// TwinCAT 3 PLC project Library
// Title: lcls-twincat-common-components
// Company: SLAC
// ProjectVersion: 4.0.0
// ProgramVersion: 3.1.4026.17
// libraries:
//   LCLS General, * (SLAC)
//   LCLS_Tc_Motion, * (SLAC - LCLS)
//   LCLS_Tc_DevAbs, * (SLAC - LCLS)
//   lcls-twincat-physics, * (SLAC)
//   PMPS, * (SLAC - LCLS)
//   Tc2_MC2, * (Beckhoff Automation GmbH)
//   Tc2_SerialCom, * (Beckhoff Automation GmbH)
//   Tc2_Standard, * (Beckhoff Automation GmbH)
//   Tc2_Utilities, * (Beckhoff Automation GmbH)
//   Tc3_JsonXml, * (Beckhoff Automation GmbH)
//   Tc3_Module, * (Beckhoff Automation GmbH)
//   TcUnit, * (www.tcunit.org)
// project tree:
//   Devices/ATM/ E_ATM_States.TcDUT, FB_ATM.TcPOU
//   Devices/LIC/ E_LIC_States.TcDUT, FB_LIC.TcPOU
//   Devices/PPM/ E_PPM_States.TcDUT, FB_PPM.TcPOU, FB_PPM_Gige.TcPOU, FB_PPM_PowerMeter.TcPOU
//   Devices/REF/ E_REF_States.TcDUT, FB_REF.TcPOU, FB_REF_Laser.TcPOU
//   Devices/SATT/ E_SXR_SATT_Position.TcDUT, FB_AttenuatorElementDensity.TcPOU, FB_SATT_FilterConfig.TcPOU, FB_SXR_SATT_Stage.TcPOU, ST_SATT_Filter.TcDUT
//   Devices/SLITS/ E_SlitsBlade.TcDUT, FB_SLITS.TcPOU, FB_SLITS_POWER.TcPOU
//   Devices/WFS/ E_WFS_States.TcDUT, FB_WFS.TcPOU
//   Devices/GBS/ E_GBS_States.TcDUT, FB_GBS.TcPOU
//   Devices/IPM/ E_IPM_States.TcDUT, FB_IPM.TcPOU
//   Devices/XPIM/ E_XPIM_Filters.TcDUT, E_XPIM_States.TcDUT, FB_XPIM.TcPOU, FB_XPIM_FilterWheel.TcPOU, FB_XPIM_LED.TcPOU, FB_XPIM_Opal.TcPOU
//   / PlcTask.TcTTO
//   POUs/ FB_CC_TempSensor.TcPOU, FB_CC_InternalStateConfig.TcPOU, FB_CC_StateDefaultsConfig.TcPOU, FB_CC_StatePMPSConfig.TcPOU, FB_FDQ_FlowMeter.TcPOU, FB_XTES_Flowswitch.TcPOU
//   Tests/ FB_ATMTest.TcPOU, FB_CC_TempSensorTest.TcPOU, FB_GBSTest.TcPOU, FB_IPMTest.TcPOU, FB_SATTTest.TcPOU, FB_LICTest.TcPOU, FB_PPMTest.TcPOU, FB_REFTest.TcPOU, FB_SLITS_POWERTest.TcPOU, FB_WFSTest.TcPOU, FB_XPIMTest.TcPOU, PRG_TEST.TcPOU
//   Tests/Helpers/ FB_PMPSJsonTestHelper.TcPOU, FB_CC_PMPSTestSetup.TcPOU
//   Version/ Global_Version.TcGVL
// real-time tasks:
//   TASK PlcTask: cycle T#10ms, priority 20, ADS port 350
// motion (NC):
//   TASK NC-Task 1 SAF: cycle T#2ms, priority 4, ADS port 501
//   TASK NC-Task 1 SVB: cycle T#10ms, priority 8, ADS port 511
//   AXIS IPM_Y (id 13)
//   AXIS GBS_Y (id 12)
//   AXIS ATM_Y (id 1)
//     OtherSettings: AllowMotionCmdToSlave=true
//     encoder EncType=1
//     drive DrvType=5
//       Analog: TorqueSetpointScale=10, ScaleFactorActTorque=0.1
//       TimeComp: TaskDelayCycles=1
//     controller CtrType=1
//       CtrPara: PriorControlFactor=1
//         Observer: BandWidth=20
//   AXIS LIC_Y (id 2)
//     OtherSettings: AllowMotionCmdToSlave=true
//     encoder EncType=1
//     drive DrvType=5
//       Analog: TorqueSetpointScale=10, ScaleFactorActTorque=0.1
//       TimeComp: TaskDelayCycles=1
//     controller CtrType=1
//       CtrPara: PriorControlFactor=1
//         Observer: BandWidth=20
//   AXIS PPM_Y (id 3)
//     OtherSettings: AllowMotionCmdToSlave=true
//     encoder EncType=1
//     drive DrvType=5
//       Analog: TorqueSetpointScale=10, ScaleFactorActTorque=0.1
//       TimeComp: TaskDelayCycles=1
//     controller CtrType=1
//       CtrPara: PriorControlFactor=1
//         Observer: BandWidth=20
//   AXIS REF_Y (id 4)
//     OtherSettings: AllowMotionCmdToSlave=true
//     encoder EncType=1
//     drive DrvType=5
//       Analog: TorqueSetpointScale=10, ScaleFactorActTorque=0.1
//       TimeComp: TaskDelayCycles=1
//     controller CtrType=1
//       CtrPara: PriorControlFactor=1
//         Observer: BandWidth=20
//   AXIS SATT_Y (id 7)
//     OtherSettings: AllowMotionCmdToSlave=true
//     encoder EncType=1
//     drive DrvType=5
//       Analog: TorqueSetpointScale=10, ScaleFactorActTorque=0.1
//     controller CtrType=1
//       CtrPara: PriorControlFactor=1
//         Observer: BandWidth=20
//   AXIS WFS_Y (id 5)
//     OtherSettings: AllowMotionCmdToSlave=true
//     encoder EncType=1
//     drive DrvType=5
//       Analog: TorqueSetpointScale=10, ScaleFactorActTorque=0.1
//       TimeComp: TaskDelayCycles=1
//     controller CtrType=1
//       CtrPara: PriorControlFactor=1
//         Observer: BandWidth=20
//   AXIS XPIM_Y (id 6)
//     OtherSettings: AllowMotionCmdToSlave=true
//     encoder EncType=1
//     drive DrvType=5
//       Analog: TorqueSetpointScale=10, ScaleFactorActTorque=0.1
//       TimeComp: TaskDelayCycles=1
//     controller CtrType=1
//       CtrPara: PriorControlFactor=1
//         Observer: BandWidth=20
//   AXIS SLIT_Bottom (id 9)
//   AXIS SLIT_North (id 10)
//   AXIS SLIT_South (id 11)
//   AXIS SLIT_Top (id 8)
//     OtherSettings: AllowMotionCmdToSlave=true
//     encoder EncType=1
//     drive DrvType=5
//       Analog: TorqueSetpointScale=10, ScaleFactorActTorque=0.1
//       TimeComp: TaskDelayCycles=1
//     controller CtrType=1
//       CtrPara: PriorControlFactor=1
//         Observer: BandWidth=20
// variable links:
//   Library Instance <-> NC-Task 1 SAF/Axes/ATM_Y
//     PlcTask Inputs/PRG_TEST.fbATMTest.axRef[2].NcToPlc <-> Outputs/ToPlc
//     PlcTask Outputs/PRG_TEST.fbATMTest.axRef[2].PlcToNc <-> Inputs/FromPlc
//   Library Instance <-> NC-Task 1 SAF/Axes/GBS_Y
//     PlcTask Inputs/PRG_TEST.fbGBSTest.axRef.NcToPlc <-> Outputs/ToPlc
//     PlcTask Outputs/PRG_TEST.fbGBSTest.axRef.PlcToNc <-> Inputs/FromPlc
//   Library Instance <-> NC-Task 1 SAF/Axes/IPM_Y
//     PlcTask Inputs/PRG_TEST.fbIPMTest.axRef[2].NcToPlc <-> Outputs/ToPlc
//     PlcTask Outputs/PRG_TEST.fbIPMTest.axRef[2].PlcToNc <-> Inputs/FromPlc
//   Library Instance <-> NC-Task 1 SAF/Axes/LIC_Y
//     PlcTask Inputs/PRG_TEST.fbLICTest.axRef.NcToPlc <-> Outputs/ToPlc
//     PlcTask Outputs/PRG_TEST.fbLICTest.axRef.PlcToNc <-> Inputs/FromPlc
//   Library Instance <-> NC-Task 1 SAF/Axes/PPM_Y
//     PlcTask Inputs/PRG_TEST.fbPPMTest.axRef.NcToPlc <-> Outputs/ToPlc
//     PlcTask Outputs/PRG_TEST.fbPPMTest.axRef.PlcToNc <-> Inputs/FromPlc
//   Library Instance <-> NC-Task 1 SAF/Axes/REF_Y
//     PlcTask Inputs/PRG_TEST.fbREFTest.axRef[2].NcToPlc <-> Outputs/ToPlc
//     PlcTask Outputs/PRG_TEST.fbREFTest.axRef[2].PlcToNc <-> Inputs/FromPlc
//   Library Instance <-> NC-Task 1 SAF/Axes/SATT_Y
//     PlcTask Inputs/PRG_TEST.fbSATTTest.axRef.NcToPlc <-> Outputs/ToPlc
//     PlcTask Outputs/PRG_TEST.fbSATTTest.axRef.PlcToNc <-> Inputs/FromPlc
//   Library Instance <-> NC-Task 1 SAF/Axes/SLIT_Bottom
//     PlcTask Inputs/PRG_TEST.fbSlitsPowerTest.axRef[2].NcToPlc <-> Outputs/ToPlc
//     PlcTask Outputs/PRG_TEST.fbSlitsPowerTest.axRef[2].PlcToNc <-> Inputs/FromPlc
//   Library Instance <-> NC-Task 1 SAF/Axes/SLIT_North
//     PlcTask Inputs/PRG_TEST.fbSlitsPowerTest.axRef[3].NcToPlc <-> Outputs/ToPlc
//     PlcTask Outputs/PRG_TEST.fbSlitsPowerTest.axRef[3].PlcToNc <-> Inputs/FromPlc
//   Library Instance <-> NC-Task 1 SAF/Axes/SLIT_South
//     PlcTask Inputs/PRG_TEST.fbSlitsPowerTest.axRef[4].NcToPlc <-> Outputs/ToPlc
//     PlcTask Outputs/PRG_TEST.fbSlitsPowerTest.axRef[4].PlcToNc <-> Inputs/FromPlc
//   Library Instance <-> NC-Task 1 SAF/Axes/SLIT_Top
//     PlcTask Inputs/PRG_TEST.fbSlitsPowerTest.axRef[1].NcToPlc <-> Outputs/ToPlc
//     PlcTask Outputs/PRG_TEST.fbSlitsPowerTest.axRef[1].PlcToNc <-> Inputs/FromPlc
//   Library Instance <-> NC-Task 1 SAF/Axes/WFS_Y
//     PlcTask Inputs/PRG_TEST.fbWFSTest.axRef[2].NcToPlc <-> Outputs/ToPlc
//     PlcTask Outputs/PRG_TEST.fbWFSTest.axRef[2].PlcToNc <-> Inputs/FromPlc
//   Library Instance <-> NC-Task 1 SAF/Axes/XPIM_Y
//     PlcTask Inputs/PRG_TEST.fbXPIMTest.axRef[3].NcToPlc <-> Outputs/ToPlc
//     PlcTask Outputs/PRG_TEST.fbXPIMTest.axRef[3].PlcToNc <-> Inputs/FromPlc

CONFIGURATION Library
    RESOURCE PLC ON TwinCAT3
        TASK PlcTask(INTERVAL := T#10ms, PRIORITY := 20);
        PROGRAM PRG_TEST WITH PlcTask : PRG_TEST;
    END_RESOURCE
END_CONFIGURATION

// ---- Devices/ATM/E_ATM_States.TcDUT
{attribute 'qualified_only'}
TYPE E_ATM_States :
(
    Unknown := 0,
    OUT := 1,
    TARGET1 := 2,
    TARGET2 := 3,
    TARGET3 := 4,
    TARGET4 := 5,
    TARGET5 := 6,
    TARGET6 := 7,
    TARGET7 := 8
) UINT;
END_TYPE

// ---- Devices/LIC/E_LIC_States.TcDUT
{attribute 'qualified_only'}
TYPE E_LIC_States :
(
    Unknown := 0,
    OUT := 1,
    MIRROR1 := 2,
    MIRROR2 := 3,
    TARGET := 4
) UINT;
END_TYPE

// ---- Devices/PPM/E_PPM_States.TcDUT
{attribute 'qualified_only'}
TYPE E_PPM_States :
(
    Unknown := 0,
    OUT := 1,
    POWERMETER := 2,
    YAG1 := 3,
    YAG2 := 4
) UINT;
END_TYPE

// ---- Devices/REF/E_REF_States.TcDUT
(* REF state-select enum. UINT-typed so REFERENCE TO E_REF_States
   is bridge-compatible with the ND mover's REFERENCE TO UINT. *)
{attribute 'qualified_only'}
{attribute 'strict'}
TYPE E_REF_States :
(
    UNKNOWN := 0,
    OUT     := 1,
    IN      := 2
) UINT;
END_TYPE

// ---- Devices/SATT/E_SXR_SATT_Position.TcDUT
{attribute 'qualified_only'}
TYPE E_SXR_SATT_Position :
(
    UNKNOWN := 0, // UNKNOWN must be in slot 0 or the FB breaks
    OUT := 1, // OUT at slot 1 is a convention
    FILTER1 := 2,
    FILTER2 := 3,
    FILTER3 := 4,
    FILTER4 := 5,
    FILTER5 := 6,
    FILTER6 := 7,
    FILTER7 := 8,
    FILTER8 := 9
) UINT;
END_TYPE

// ---- Devices/SATT/ST_SATT_Filter.TcDUT
TYPE ST_SATT_Filter :
STRUCT
    {attribute 'pytmc' := '
        pv: MATERIAL
        io: input
        field: DESC Filter material name
    '}
    sFilterMaterial : STRING;

    {attribute 'pytmc' := '
        pv: THICKNESS
        io: input
        field: DESC Filter material thickness
        field: EGU um
    '}
    fFilterThickness_um : LREAL;
END_STRUCT
END_TYPE

// ---- Devices/SLITS/E_SlitsBlade.TcDUT
(* Blade index into the four-element slit motion-stage array
   (Top / Bottom / North / South). Values 1..4 match the array bounds. *)
{attribute 'qualified_only'}
{attribute 'strict'}
TYPE E_SlitsBlade :
(
    TOP    := 1,
    BOTTOM := 2,
    NORTH  := 3,
    SOUTH  := 4
) UDINT;
END_TYPE

// ---- Devices/WFS/E_WFS_States.TcDUT
{attribute 'qualified_only'}
TYPE E_WFS_States :
(
    Unknown := 0,
    OUT := 1,
    TARGET1 := 2,
    TARGET2 := 3,
    TARGET3 := 4,
    TARGET4 := 5,
    TARGET5 := 6
) UINT;
END_TYPE

// ---- Devices/GBS/E_GBS_States.TcDUT
{attribute 'qualified_only'}
TYPE E_GBS_States :
(
    Unknown := 0,
    OUT := 1,
    TARGET1a := 2,
    TARGET1b := 3,
    TARGET2a := 4,
    TARGET2b := 5,
    TARGET3a := 6,
    TARGET3b := 7,
    TARGET4 := 8,
    TARGET5 := 9,
    TARGET6 := 10
) UINT;
END_TYPE

// ---- Devices/IPM/E_IPM_States.TcDUT
{attribute 'qualified_only'}
TYPE E_IPM_States :
(
    Unknown := 0,
    OUT := 1,
    TARGET1 := 2,
    TARGET2 := 3,
    TARGET3 := 4,
    TARGET4 := 5
) UINT;
END_TYPE

// ---- Devices/XPIM/E_XPIM_Filters.TcDUT
{attribute 'qualified_only'}
TYPE E_XPIM_Filters :
(
    Unknown := 0,
    T50 := 1,
    T25 := 2,
    T10 := 3,
    T5 := 4,
    T1 := 5,
    T100 := 6
) UINT;
END_TYPE

// ---- Devices/XPIM/E_XPIM_States.TcDUT
{attribute 'qualified_only'}
TYPE E_XPIM_States :
(
    Unknown := 0,
    OUT := 1,
    YAG := 2,
    DIAMOND := 3,
    RETICLE := 4
) UINT;
END_TYPE

// ---- Version/Global_Version.TcGVL
{attribute 'TcGenerated'}
{attribute 'no-analysis'}
{attribute 'linkalways'}
// This function has been automatically generated from the project information.
VAR_GLOBAL CONSTANT
    {attribute 'const_non_replaced'}
    stLibVersion_lcls_twincat_common_components : ST_LibVersion := (iMajor := 4, iMinor := 0, iBuild := 0, iRevision := 0, nFlags := 1, sVersion := '4.0.0');
END_VAR

// ---- Tests/PRG_TEST.TcPOU
{attribute 'analysis' := '-33'}
PROGRAM PRG_TEST
VAR
    (* Seeds PMPS_GVL.BP_jsonDoc with the fake test PMPS DB in before any test FB body runs. *)
    fbPmpsTestSetup: FB_CC_PMPSTestSetup;
    fbATMTest: FB_ATMTest;
    fbGBSTest: FB_GBSTest;
    fbIPMTest: FB_IPMTest;
    fbLICTest: FB_LICTest;
    fbPPMTest: FB_PPMTest;
    fbREFTest: FB_REFTest;
    fbSATTTest: FB_SATTTest;
    fbSlitsPowerTest: FB_SLITS_POWERTest;
    fbWFSTest: FB_WFSTest;
    fbXPIMTest: FB_XPIMTest;
    fbCCTempSensorTest: FB_CC_TempSensorTest;


END_VAR

// Run the tests
TcUnit.RUN();

END_PROGRAM

// ---- Tests/Helpers/FB_CC_PMPSTestSetup.TcPOU

(*
    One-shot PMPS fake-DB seeder for the CC test suite. Mirrors
    LCLS_Tc_Motion.FB_PMPSTestSetup: one FB_PMPSJsonTestHelperEx
    instance per device, first call uses bNewDoc := TRUE, the rest
    use bNewDoc := FALSE so the document at PMPS_GVL.BP_jsonDoc
    accumulates every test device:

        { "TST:ATM": { "TST:ATM-TRANSITION": {...}, ... },
          "TST:LIC": { ... }, ... }

    Only sPmpsState is populated per row. The helper fills the rest
    of the JSON shape with default-zero values, which is enough for
    the wiring smoke tests to look up state keys and request a move.
    Tests that need richer beam params (rate, beam class, eV range,
    reactive temperature) set them on the relevant astParams_XXX
    entries before this FB ticks, or extend it.

    The seeding runs once in CallAfterInit, before any test suite
    body executes. The cyclic body is empty: no scheduling order
    dependency between this FB and the test FBs.

    Single point of truth: PMPS_GVL.BP_jsonDoc is global and test
    FBs run concurrently. Seeding stays here so per-device writes
    cannot race on the same cycle.
*)
{attribute 'call_after_init'}
{attribute 'analysis' := '-33'}
FUNCTION_BLOCK FB_CC_PMPSTestSetup
VAR
    (* All devices use the local FB_PMPSJsonTestHelper: it serializes the
       seeded nRequestAssertionID into the DB 'id' (so each state gets a
       unique assertion ID) and serializes nTempSP into reactive_temp
       (needed by SATT/SLITS RTD thresholds). *)
    fbJsonHelper_ATM   : FB_PMPSJsonTestHelper;
    fbJsonHelper_LIC   : FB_PMPSJsonTestHelper;
    fbJsonHelper_PPM   : FB_PMPSJsonTestHelper;
    fbJsonHelper_REF   : FB_PMPSJsonTestHelper;
    fbJsonHelper_GBS   : FB_PMPSJsonTestHelper;
    fbJsonHelper_IPM   : FB_PMPSJsonTestHelper;
    fbJsonHelper_WFS   : FB_PMPSJsonTestHelper;
    fbJsonHelper_XPIM  : FB_PMPSJsonTestHelper;
    fbJsonHelper_SATT  : FB_PMPSJsonTestHelper;
    fbJsonHelper_SLITS : FB_PMPSJsonTestHelper;

    (* astParams_XXX[0] is the transition key; the rest are named-state
       keys in enum order. *)
    astParams_ATM   : ARRAY[0..6] OF ST_DbStateParams;
    astParams_LIC   : ARRAY[0..4] OF ST_DbStateParams;
    astParams_PPM   : ARRAY[0..4] OF ST_DbStateParams;
    astParams_REF   : ARRAY[0..2] OF ST_DbStateParams;
    astParams_GBS   : ARRAY[0..10] OF ST_DbStateParams;
    astParams_IPM   : ARRAY[0..5] OF ST_DbStateParams;
    astParams_WFS   : ARRAY[0..6] OF ST_DbStateParams;
    astParams_XPIM  : ARRAY[0..5] OF ST_DbStateParams;
    astParams_SATT  : ARRAY[0..0] OF ST_DbStateParams;
    astParams_SLITS : ARRAY[0..0] OF ST_DbStateParams;
END_VAR


(* Seeding runs once at instantiation in CallAfterInit; body is a no-op. *)

{attribute 'call_after_init'}
METHOD CallAfterInit

(* ---- TST:ATM ---- *)
astParams_ATM[0].sPmpsState                  := 'TST:ATM-TRANSITION';
astParams_ATM[0].nRequestAssertionID         := 100;
astParams_ATM[0].stReactiveParams.nTempSP   := 30;
astParams_ATM[0].stBeamParams.nBeamClass     := 2#0000_1000;
astParams_ATM[0].stBeamParams.neVRange       := 2#1111_1111_1111_1111_1111_1111_1111_1111;
astParams_ATM[0].stBeamParams.nRate          := 1;
astParams_ATM[0].stBeamParams.nTran          := 0;
astParams_ATM[0].stBeamParams.nMachineMode   := 1;

astParams_ATM[1].sPmpsState                  := 'TST:ATM-OUT';
astParams_ATM[1].nRequestAssertionID         := 101;
astParams_ATM[1].stReactiveParams.nTempSP   := 30;
astParams_ATM[1].stBeamParams.nBeamClass     := 2#0000_0001;
astParams_ATM[1].stBeamParams.neVRange       := 2#1111_1111_1111_1111_1111_1111_1111_1111;
astParams_ATM[1].stBeamParams.nRate          := 10;
astParams_ATM[1].stBeamParams.nTran          := 12;
astParams_ATM[1].stBeamParams.nMachineMode   := 2;

astParams_ATM[2].sPmpsState                  := 'TST:ATM-TARGET1';
astParams_ATM[2].nRequestAssertionID         := 102;
astParams_ATM[2].stReactiveParams.nTempSP   := 30;
astParams_ATM[2].stBeamParams.nBeamClass     := 2#0000_0010;
astParams_ATM[2].stBeamParams.neVRange       := 2#1111_1111_1111_1111_1111_1111_1111_1111;
astParams_ATM[2].stBeamParams.nRate          := 50;
astParams_ATM[2].stBeamParams.nTran          := 8;
astParams_ATM[2].stBeamParams.nMachineMode   := 1;

astParams_ATM[3].sPmpsState                  := 'TST:ATM-TARGET2';
astParams_ATM[3].nRequestAssertionID         := 103;
astParams_ATM[3].stReactiveParams.nTempSP   := 30;
astParams_ATM[3].stBeamParams.nBeamClass     := 2#0000_0100;
astParams_ATM[3].stBeamParams.neVRange       := 2#1111_1111_1111_1111_1111_1111_1111_1111;
astParams_ATM[3].stBeamParams.nRate          := 50;
astParams_ATM[3].stBeamParams.nTran          := 8;
astParams_ATM[3].stBeamParams.nMachineMode   := 1;

astParams_ATM[4].sPmpsState                  := 'TST:ATM-TARGET3';
astParams_ATM[4].nRequestAssertionID         := 104;
astParams_ATM[4].stReactiveParams.nTempSP   := 30;
astParams_ATM[4].stBeamParams.nBeamClass     := 2#0001_0000;
astParams_ATM[4].stBeamParams.neVRange       := 2#1111_1111_1111_1111_1111_1111_1111_1111;
astParams_ATM[4].stBeamParams.nRate          := 50;
astParams_ATM[4].stBeamParams.nTran          := 8;
astParams_ATM[4].stBeamParams.nMachineMode   := 1;

astParams_ATM[5].sPmpsState                  := 'TST:ATM-TARGET4';
astParams_ATM[5].nRequestAssertionID         := 105;
astParams_ATM[5].stReactiveParams.nTempSP   := 30;
astParams_ATM[5].stBeamParams.nBeamClass     := 2#0010_0000;
astParams_ATM[5].stBeamParams.neVRange       := 2#1111_1111_1111_1111_1111_1111_1111_1111;
astParams_ATM[5].stBeamParams.nRate          := 50;
astParams_ATM[5].stBeamParams.nTran          := 8;
astParams_ATM[5].stBeamParams.nMachineMode   := 1;

astParams_ATM[6].sPmpsState                  := 'TST:ATM-TARGET5';
astParams_ATM[6].nRequestAssertionID         := 106;
astParams_ATM[6].stReactiveParams.nTempSP   := 30;
astParams_ATM[6].stBeamParams.nBeamClass     := 2#0100_0000;
astParams_ATM[6].stBeamParams.neVRange       := 2#1111_1111_1111_1111_1111_1111_1111_1111;
astParams_ATM[6].stBeamParams.nRate          := 50;
astParams_ATM[6].stBeamParams.nTran          := 8;
astParams_ATM[6].stBeamParams.nMachineMode   := 1;

(* ---- TST:LIC ---- *)
astParams_LIC[0].sPmpsState                  := 'TST:LIC-TRANSITION';
astParams_LIC[0].nRequestAssertionID         := 200;
astParams_LIC[0].stBeamParams.nBeamClass     := 2#0000_1000;
astParams_LIC[0].stBeamParams.neVRange       := 2#1111_1111_1111_1111_1111_1111_1111_1111;
astParams_LIC[0].stBeamParams.nRate          := 1;
astParams_LIC[0].stBeamParams.nTran          := 0;
astParams_LIC[0].stBeamParams.nMachineMode   := 1;

astParams_LIC[1].sPmpsState                  := 'TST:LIC-OUT';
astParams_LIC[1].nRequestAssertionID         := 201;
astParams_LIC[1].stBeamParams.nBeamClass     := 2#0000_0001;
astParams_LIC[1].stBeamParams.neVRange       := 2#1111_1111_1111_1111_1111_1111_1111_1111;
astParams_LIC[1].stBeamParams.nRate          := 10;
astParams_LIC[1].stBeamParams.nTran          := 12;
astParams_LIC[1].stBeamParams.nMachineMode   := 2;

astParams_LIC[2].sPmpsState                  := 'TST:LIC-MIRROR1';
astParams_LIC[2].nRequestAssertionID         := 202;
astParams_LIC[2].stBeamParams.nBeamClass     := 2#0000_0010;
astParams_LIC[2].stBeamParams.neVRange       := 2#1111_1111_1111_1111_1111_1111_1111_1111;
astParams_LIC[2].stBeamParams.nRate          := 50;
astParams_LIC[2].stBeamParams.nTran          := 8;
astParams_LIC[2].stBeamParams.nMachineMode   := 1;

astParams_LIC[3].sPmpsState                  := 'TST:LIC-MIRROR2';
astParams_LIC[3].nRequestAssertionID         := 203;
astParams_LIC[3].stBeamParams.nBeamClass     := 2#0000_0100;
astParams_LIC[3].stBeamParams.neVRange       := 2#1111_1111_1111_1111_1111_1111_1111_1111;
astParams_LIC[3].stBeamParams.nRate          := 50;
astParams_LIC[3].stBeamParams.nTran          := 8;
astParams_LIC[3].stBeamParams.nMachineMode   := 1;

astParams_LIC[4].sPmpsState                  := 'TST:LIC-TARGET';
astParams_LIC[4].nRequestAssertionID         := 204;
astParams_LIC[4].stBeamParams.nBeamClass     := 2#0001_0000;
astParams_LIC[4].stBeamParams.neVRange       := 2#1111_1111_1111_1111_1111_1111_1111_1111;
astParams_LIC[4].stBeamParams.nRate          := 50;
astParams_LIC[4].stBeamParams.nTran          := 8;
astParams_LIC[4].stBeamParams.nMachineMode   := 1;

(* ---- TST:PPM ---- *)
astParams_PPM[0].sPmpsState                  := 'TST:PPM-TRANSITION';
astParams_PPM[0].stReactiveParams.nTempSP   := 30;
astParams_PPM[0].nRequestAssertionID         := 300;
astParams_PPM[0].stBeamParams.nBeamClass     := 2#0000_1000;
astParams_PPM[0].stBeamParams.neVRange       := 2#1111_1111_1111_1111_1111_1111_1111_1111;
astParams_PPM[0].stBeamParams.nRate          := 1;
astParams_PPM[0].stBeamParams.nTran          := 0;
astParams_PPM[0].stBeamParams.nMachineMode   := 1;

astParams_PPM[1].sPmpsState                  := 'TST:PPM-OUT';
astParams_PPM[1].stReactiveParams.nTempSP   := 30;
astParams_PPM[1].nRequestAssertionID         := 301;
astParams_PPM[1].stBeamParams.nBeamClass     := 2#0000_0001;
astParams_PPM[1].stBeamParams.neVRange       := 2#1111_1111_1111_1111_1111_1111_1111_1111;
astParams_PPM[1].stBeamParams.nRate          := 10;
astParams_PPM[1].stBeamParams.nTran          := 12;
astParams_PPM[1].stBeamParams.nMachineMode   := 2;

astParams_PPM[2].sPmpsState                  := 'TST:PPM-POWERMETER';
astParams_PPM[2].stReactiveParams.nTempSP   := 30;
astParams_PPM[2].nRequestAssertionID         := 302;
astParams_PPM[2].stBeamParams.nBeamClass     := 2#0000_0010;
astParams_PPM[2].stBeamParams.neVRange       := 2#1111_1111_1111_1111_1111_1111_1111_1111;
astParams_PPM[2].stBeamParams.nRate          := 50;
astParams_PPM[2].stBeamParams.nTran          := 8;
astParams_PPM[2].stBeamParams.nMachineMode   := 1;

astParams_PPM[3].sPmpsState                  := 'TST:PPM-YAG1';
astParams_PPM[3].stReactiveParams.nTempSP   := 30;
astParams_PPM[3].nRequestAssertionID         := 303;
astParams_PPM[3].stBeamParams.nBeamClass     := 2#0000_0100;
astParams_PPM[3].stBeamParams.neVRange       := 2#1111_1111_1111_1111_1111_1111_1111_1111;
astParams_PPM[3].stBeamParams.nRate          := 50;
astParams_PPM[3].stBeamParams.nTran          := 8;
astParams_PPM[3].stBeamParams.nMachineMode   := 1;

astParams_PPM[4].sPmpsState                  := 'TST:PPM-YAG2';
astParams_PPM[4].stReactiveParams.nTempSP   := 30;
astParams_PPM[4].nRequestAssertionID         := 304;
astParams_PPM[4].stBeamParams.nBeamClass     := 2#0001_0000;
astParams_PPM[4].stBeamParams.neVRange       := 2#1111_1111_1111_1111_1111_1111_1111_1111;
astParams_PPM[4].stBeamParams.nRate          := 50;
astParams_PPM[4].stBeamParams.nTran          := 8;
astParams_PPM[4].stBeamParams.nMachineMode   := 1;

(* ---- TST:REF ---- *)
astParams_REF[0].sPmpsState                  := 'TST:REF-TRANSITION';
astParams_REF[0].nRequestAssertionID         := 600;
astParams_REF[0].stBeamParams.nBeamClass     := 2#0000_1000;
astParams_REF[0].stBeamParams.neVRange       := 2#1111_1111_1111_1111_1111_1111_1111_1111;
astParams_REF[0].stBeamParams.nRate          := 1;
astParams_REF[0].stBeamParams.nTran          := 0;
astParams_REF[0].stBeamParams.nMachineMode   := 1;

astParams_REF[1].sPmpsState                  := 'TST:REF-OUT';
astParams_REF[1].nRequestAssertionID         := 601;
astParams_REF[1].stBeamParams.nBeamClass     := 2#0000_0001;
astParams_REF[1].stBeamParams.neVRange       := 2#1111_1111_1111_1111_1111_1111_1111_1111;
astParams_REF[1].stBeamParams.nRate          := 10;
astParams_REF[1].stBeamParams.nTran          := 12;
astParams_REF[1].stBeamParams.nMachineMode   := 2;

astParams_REF[2].sPmpsState                  := 'TST:REF-IN';
astParams_REF[2].nRequestAssertionID         := 602;
astParams_REF[2].stBeamParams.nBeamClass     := 2#1000_0000;
astParams_REF[2].stBeamParams.neVRange       := 2#1111_1111_1111_1111_1111_1111_1111_1111;
astParams_REF[2].stBeamParams.nRate          := 110;
astParams_REF[2].stBeamParams.nTran          := 12.5;
astParams_REF[2].stBeamParams.nMachineMode   := 1;

(* ---- TST:GBS ---- *)
astParams_GBS[0].sPmpsState                  := 'TST:GBS-TRANSITION';
astParams_GBS[0].nRequestAssertionID         := 700;
astParams_GBS[0].stBeamParams.nBeamClass     := 2#0000_1000;
astParams_GBS[0].stBeamParams.neVRange       := 2#1111_1111_1111_1111_1111_1111_1111_1111;
astParams_GBS[0].stBeamParams.nRate          := 1;
astParams_GBS[0].stBeamParams.nTran          := 0;
astParams_GBS[0].stBeamParams.nMachineMode   := 1;

astParams_GBS[1].sPmpsState                  := 'TST:GBS-OUT';
astParams_GBS[1].nRequestAssertionID         := 701;
astParams_GBS[1].stBeamParams.nBeamClass     := 2#0000_0001;
astParams_GBS[1].stBeamParams.neVRange       := 2#1111_1111_1111_1111_1111_1111_1111_1111;
astParams_GBS[1].stBeamParams.nRate          := 10;
astParams_GBS[1].stBeamParams.nTran          := 12;
astParams_GBS[1].stBeamParams.nMachineMode   := 2;

astParams_GBS[2].sPmpsState                  := 'TST:GBS-TARGET1a';
astParams_GBS[2].nRequestAssertionID         := 702;
astParams_GBS[2].stBeamParams.nBeamClass     := 2#0000_0010;
astParams_GBS[2].stBeamParams.neVRange       := 2#1111_1111_1111_1111_1111_1111_1111_1111;
astParams_GBS[2].stBeamParams.nRate          := 50;
astParams_GBS[2].stBeamParams.nTran          := 8;
astParams_GBS[2].stBeamParams.nMachineMode   := 1;

astParams_GBS[3].sPmpsState                  := 'TST:GBS-TARGET1b';
astParams_GBS[3].nRequestAssertionID         := 703;
astParams_GBS[3].stBeamParams.nBeamClass     := 2#0000_0100;
astParams_GBS[3].stBeamParams.neVRange       := 2#1111_1111_1111_1111_1111_1111_1111_1111;
astParams_GBS[3].stBeamParams.nRate          := 50;
astParams_GBS[3].stBeamParams.nTran          := 8;
astParams_GBS[3].stBeamParams.nMachineMode   := 1;

astParams_GBS[4].sPmpsState                  := 'TST:GBS-TARGET2a';
astParams_GBS[4].nRequestAssertionID         := 704;
astParams_GBS[4].stBeamParams.nBeamClass     := 2#0001_0000;
astParams_GBS[4].stBeamParams.neVRange       := 2#1111_1111_1111_1111_1111_1111_1111_1111;
astParams_GBS[4].stBeamParams.nRate          := 50;
astParams_GBS[4].stBeamParams.nTran          := 8;
astParams_GBS[4].stBeamParams.nMachineMode   := 1;

astParams_GBS[5].sPmpsState                  := 'TST:GBS-TARGET2b';
astParams_GBS[5].nRequestAssertionID         := 705;
astParams_GBS[5].stBeamParams.nBeamClass     := 2#0010_0000;
astParams_GBS[5].stBeamParams.neVRange       := 2#1111_1111_1111_1111_1111_1111_1111_1111;
astParams_GBS[5].stBeamParams.nRate          := 50;
astParams_GBS[5].stBeamParams.nTran          := 8;
astParams_GBS[5].stBeamParams.nMachineMode   := 1;

astParams_GBS[6].sPmpsState                  := 'TST:GBS-TARGET3a';
astParams_GBS[6].nRequestAssertionID         := 706;
astParams_GBS[6].stBeamParams.nBeamClass     := 2#0100_0000;
astParams_GBS[6].stBeamParams.neVRange       := 2#1111_1111_1111_1111_1111_1111_1111_1111;
astParams_GBS[6].stBeamParams.nRate          := 50;
astParams_GBS[6].stBeamParams.nTran          := 8;
astParams_GBS[6].stBeamParams.nMachineMode   := 1;

astParams_GBS[7].sPmpsState                  := 'TST:GBS-TARGET3b';
astParams_GBS[7].nRequestAssertionID         := 707;
astParams_GBS[7].stBeamParams.nBeamClass     := 2#1000_0000;
astParams_GBS[7].stBeamParams.neVRange       := 2#1111_1111_1111_1111_1111_1111_1111_1111;
astParams_GBS[7].stBeamParams.nRate          := 50;
astParams_GBS[7].stBeamParams.nTran          := 8;
astParams_GBS[7].stBeamParams.nMachineMode   := 1;

astParams_GBS[8].sPmpsState                  := 'TST:GBS-TARGET4';
astParams_GBS[8].nRequestAssertionID         := 708;
astParams_GBS[8].stBeamParams.nBeamClass     := 2#0000_0010;
astParams_GBS[8].stBeamParams.neVRange       := 2#1111_1111_1111_1111_1111_1111_1111_1111;
astParams_GBS[8].stBeamParams.nRate          := 50;
astParams_GBS[8].stBeamParams.nTran          := 8;
astParams_GBS[8].stBeamParams.nMachineMode   := 1;

astParams_GBS[9].sPmpsState                  := 'TST:GBS-TARGET5';
astParams_GBS[9].nRequestAssertionID         := 709;
astParams_GBS[9].stBeamParams.nBeamClass     := 2#0000_0100;
astParams_GBS[9].stBeamParams.neVRange       := 2#1111_1111_1111_1111_1111_1111_1111_1111;
astParams_GBS[9].stBeamParams.nRate          := 50;
astParams_GBS[9].stBeamParams.nTran          := 8;
astParams_GBS[9].stBeamParams.nMachineMode   := 1;

astParams_GBS[10].sPmpsState                 := 'TST:GBS-TARGET6';
astParams_GBS[10].nRequestAssertionID        := 710;
astParams_GBS[10].stBeamParams.nBeamClass    := 2#0001_0000;
astParams_GBS[10].stBeamParams.neVRange      := 2#1111_1111_1111_1111_1111_1111_1111_1111;
astParams_GBS[10].stBeamParams.nRate         := 50;
astParams_GBS[10].stBeamParams.nTran         := 8;
astParams_GBS[10].stBeamParams.nMachineMode  := 1;

(* In-beam RTD setpoint for FB_GBSTest temp-FFO wiring: the two RTDs
   fault when the reading exceeds nTempSP and are vetoed while OUT. *)
astParams_GBS[0].stReactiveParams.nTempSP    := 30;
astParams_GBS[1].stReactiveParams.nTempSP    := 30;
astParams_GBS[2].stReactiveParams.nTempSP    := 30;
astParams_GBS[3].stReactiveParams.nTempSP    := 30;
astParams_GBS[4].stReactiveParams.nTempSP    := 30;
astParams_GBS[5].stReactiveParams.nTempSP    := 30;
astParams_GBS[6].stReactiveParams.nTempSP    := 30;
astParams_GBS[7].stReactiveParams.nTempSP    := 30;
astParams_GBS[8].stReactiveParams.nTempSP    := 30;
astParams_GBS[9].stReactiveParams.nTempSP    := 30;
astParams_GBS[10].stReactiveParams.nTempSP   := 30;

(* ---- TST:IPM ---- *)
astParams_IPM[0].sPmpsState                  := 'TST:IPM-TRANSITION';
astParams_IPM[0].nRequestAssertionID         := 800;
astParams_IPM[0].stBeamParams.nBeamClass     := 2#0000_1000;
astParams_IPM[0].stBeamParams.neVRange       := 2#1111_1111_1111_1111_1111_1111_1111_1111;
astParams_IPM[0].stBeamParams.nRate          := 1;
astParams_IPM[0].stBeamParams.nTran          := 0;
astParams_IPM[0].stBeamParams.nMachineMode   := 1;

astParams_IPM[1].sPmpsState                  := 'TST:IPM-OUT';
astParams_IPM[1].nRequestAssertionID         := 801;
astParams_IPM[1].stBeamParams.nBeamClass     := 2#0000_0001;
astParams_IPM[1].stBeamParams.neVRange       := 2#1111_1111_1111_1111_1111_1111_1111_1111;
astParams_IPM[1].stBeamParams.nRate          := 10;
astParams_IPM[1].stBeamParams.nTran          := 12;
astParams_IPM[1].stBeamParams.nMachineMode   := 2;

astParams_IPM[2].sPmpsState                  := 'TST:IPM-TARGET1';
astParams_IPM[2].nRequestAssertionID         := 802;
astParams_IPM[2].stBeamParams.nBeamClass     := 2#0000_0010;
astParams_IPM[2].stBeamParams.neVRange       := 2#1111_1111_1111_1111_1111_1111_1111_1111;
astParams_IPM[2].stBeamParams.nRate          := 50;
astParams_IPM[2].stBeamParams.nTran          := 8;
astParams_IPM[2].stBeamParams.nMachineMode   := 1;

astParams_IPM[3].sPmpsState                  := 'TST:IPM-TARGET2';
astParams_IPM[3].nRequestAssertionID         := 803;
astParams_IPM[3].stBeamParams.nBeamClass     := 2#0000_0100;
astParams_IPM[3].stBeamParams.neVRange       := 2#1111_1111_1111_1111_1111_1111_1111_1111;
astParams_IPM[3].stBeamParams.nRate          := 50;
astParams_IPM[3].stBeamParams.nTran          := 8;
astParams_IPM[3].stBeamParams.nMachineMode   := 1;

astParams_IPM[4].sPmpsState                  := 'TST:IPM-TARGET3';
astParams_IPM[4].nRequestAssertionID         := 804;
astParams_IPM[4].stBeamParams.nBeamClass     := 2#0001_0000;
astParams_IPM[4].stBeamParams.neVRange       := 2#1111_1111_1111_1111_1111_1111_1111_1111;
astParams_IPM[4].stBeamParams.nRate          := 50;
astParams_IPM[4].stBeamParams.nTran          := 8;
astParams_IPM[4].stBeamParams.nMachineMode   := 1;

astParams_IPM[5].sPmpsState                  := 'TST:IPM-TARGET4';
astParams_IPM[5].nRequestAssertionID         := 805;
astParams_IPM[5].stBeamParams.nBeamClass     := 2#0010_0000;
astParams_IPM[5].stBeamParams.neVRange       := 2#1111_1111_1111_1111_1111_1111_1111_1111;
astParams_IPM[5].stBeamParams.nRate          := 50;
astParams_IPM[5].stBeamParams.nTran          := 8;
astParams_IPM[5].stBeamParams.nMachineMode   := 1;

(* ---- TST:WFS ---- *)
astParams_WFS[0].sPmpsState                  := 'TST:WFS-TRANSITION';
astParams_WFS[0].stReactiveParams.nTempSP   := 30;
astParams_WFS[0].nRequestAssertionID         := 900;
astParams_WFS[0].stBeamParams.nBeamClass     := 2#0000_1000;
astParams_WFS[0].stBeamParams.neVRange       := 2#1111_1111_1111_1111_1111_1111_1111_1111;
astParams_WFS[0].stBeamParams.nRate          := 1;
astParams_WFS[0].stBeamParams.nTran          := 0;
astParams_WFS[0].stBeamParams.nMachineMode   := 1;

astParams_WFS[1].sPmpsState                  := 'TST:WFS-OUT';
astParams_WFS[1].stReactiveParams.nTempSP   := 30;
astParams_WFS[1].nRequestAssertionID         := 901;
astParams_WFS[1].stBeamParams.nBeamClass     := 2#0000_0001;
astParams_WFS[1].stBeamParams.neVRange       := 2#1111_1111_1111_1111_1111_1111_1111_1111;
astParams_WFS[1].stBeamParams.nRate          := 10;
astParams_WFS[1].stBeamParams.nTran          := 12;
astParams_WFS[1].stBeamParams.nMachineMode   := 2;

astParams_WFS[2].sPmpsState                  := 'TST:WFS-TARGET1';
astParams_WFS[2].stReactiveParams.nTempSP   := 30;
astParams_WFS[2].nRequestAssertionID         := 902;
astParams_WFS[2].stBeamParams.nBeamClass     := 2#0000_0010;
astParams_WFS[2].stBeamParams.neVRange       := 2#1111_1111_1111_1111_1111_1111_1111_1111;
astParams_WFS[2].stBeamParams.nRate          := 50;
astParams_WFS[2].stBeamParams.nTran          := 8;
astParams_WFS[2].stBeamParams.nMachineMode   := 1;

astParams_WFS[3].sPmpsState                  := 'TST:WFS-TARGET2';
astParams_WFS[3].stReactiveParams.nTempSP   := 30;
astParams_WFS[3].nRequestAssertionID         := 903;
astParams_WFS[3].stBeamParams.nBeamClass     := 2#0000_0100;
astParams_WFS[3].stBeamParams.neVRange       := 2#1111_1111_1111_1111_1111_1111_1111_1111;
astParams_WFS[3].stBeamParams.nRate          := 50;
astParams_WFS[3].stBeamParams.nTran          := 8;
astParams_WFS[3].stBeamParams.nMachineMode   := 1;

astParams_WFS[4].sPmpsState                  := 'TST:WFS-TARGET3';
astParams_WFS[4].stReactiveParams.nTempSP   := 30;
astParams_WFS[4].nRequestAssertionID         := 904;
astParams_WFS[4].stBeamParams.nBeamClass     := 2#0001_0000;
astParams_WFS[4].stBeamParams.neVRange       := 2#1111_1111_1111_1111_1111_1111_1111_1111;
astParams_WFS[4].stBeamParams.nRate          := 50;
astParams_WFS[4].stBeamParams.nTran          := 8;
astParams_WFS[4].stBeamParams.nMachineMode   := 1;

astParams_WFS[5].sPmpsState                  := 'TST:WFS-TARGET4';
astParams_WFS[5].stReactiveParams.nTempSP   := 30;
astParams_WFS[5].nRequestAssertionID         := 905;
astParams_WFS[5].stBeamParams.nBeamClass     := 2#0010_0000;
astParams_WFS[5].stBeamParams.neVRange       := 2#1111_1111_1111_1111_1111_1111_1111_1111;
astParams_WFS[5].stBeamParams.nRate          := 50;
astParams_WFS[5].stBeamParams.nTran          := 8;
astParams_WFS[5].stBeamParams.nMachineMode   := 1;

astParams_WFS[6].sPmpsState                  := 'TST:WFS-TARGET5';
astParams_WFS[6].stReactiveParams.nTempSP   := 30;
astParams_WFS[6].nRequestAssertionID         := 906;
astParams_WFS[6].stBeamParams.nBeamClass     := 2#0100_0000;
astParams_WFS[6].stBeamParams.neVRange       := 2#1111_1111_1111_1111_1111_1111_1111_1111;
astParams_WFS[6].stBeamParams.nRate          := 50;
astParams_WFS[6].stBeamParams.nTran          := 8;
astParams_WFS[6].stBeamParams.nMachineMode   := 1;

(* ---- TST:XPIM ---- *)
astParams_XPIM[0].sPmpsState                 := 'TST:XPIM-TRANSITION';
astParams_XPIM[0].nRequestAssertionID        := 1000;
astParams_XPIM[0].stBeamParams.nBeamClass    := 2#0000_1000;
astParams_XPIM[0].stBeamParams.neVRange      := 2#1111_1111_1111_1111_1111_1111_1111_1111;
astParams_XPIM[0].stBeamParams.nRate         := 1;
astParams_XPIM[0].stBeamParams.nTran         := 0;
astParams_XPIM[0].stBeamParams.nMachineMode  := 1;

astParams_XPIM[1].sPmpsState                 := 'TST:XPIM-OUT';
astParams_XPIM[1].nRequestAssertionID        := 1001;
astParams_XPIM[1].stBeamParams.nBeamClass    := 2#0000_0001;
astParams_XPIM[1].stBeamParams.neVRange      := 2#1111_1111_1111_1111_1111_1111_1111_1111;
astParams_XPIM[1].stBeamParams.nRate         := 10;
astParams_XPIM[1].stBeamParams.nTran         := 12;
astParams_XPIM[1].stBeamParams.nMachineMode  := 2;

astParams_XPIM[2].sPmpsState                 := 'TST:XPIM-DIAMOND';
astParams_XPIM[2].nRequestAssertionID        := 1002;
astParams_XPIM[2].stBeamParams.nBeamClass    := 2#0000_0010;
astParams_XPIM[2].stBeamParams.neVRange      := 2#1111_1111_1111_1111_1111_1111_1111_1111;
astParams_XPIM[2].stBeamParams.nRate         := 50;
astParams_XPIM[2].stBeamParams.nTran         := 8;
astParams_XPIM[2].stBeamParams.nMachineMode  := 1;

astParams_XPIM[3].sPmpsState                 := 'TST:XPIM-RETICLE';
astParams_XPIM[3].nRequestAssertionID        := 1003;
astParams_XPIM[3].stBeamParams.nBeamClass    := 2#0000_0100;
astParams_XPIM[3].stBeamParams.neVRange      := 2#1111_1111_1111_1111_1111_1111_1111_1111;
astParams_XPIM[3].stBeamParams.nRate         := 50;
astParams_XPIM[3].stBeamParams.nTran         := 8;
astParams_XPIM[3].stBeamParams.nMachineMode  := 1;

astParams_XPIM[4].sPmpsState                 := 'TST:XPIM-YAG';
astParams_XPIM[4].nRequestAssertionID        := 1004;
astParams_XPIM[4].stBeamParams.nBeamClass    := 2#0001_0000;
astParams_XPIM[4].stBeamParams.neVRange      := 2#1111_1111_1111_1111_1111_1111_1111_1111;
astParams_XPIM[4].stBeamParams.nRate         := 50;
astParams_XPIM[4].stBeamParams.nTran         := 8;
astParams_XPIM[4].stBeamParams.nMachineMode  := 1;

astParams_XPIM[5].sPmpsState                 := 'TST:XPIM-POWERMETER';
astParams_XPIM[5].nRequestAssertionID        := 1005;
astParams_XPIM[5].stBeamParams.nBeamClass    := 2#0010_0000;
astParams_XPIM[5].stBeamParams.neVRange      := 2#1111_1111_1111_1111_1111_1111_1111_1111;
astParams_XPIM[5].stBeamParams.nRate         := 50;
astParams_XPIM[5].stBeamParams.nTran         := 8;
astParams_XPIM[5].stBeamParams.nMachineMode  := 1;

(* ---- AT1K4:L2SI (single reactive-temp key; the SATT filters are not
   real PMPS states, so only the RTD reactive-temperature key is
   seeded). nTempSP is the RTD fault threshold in degC: the SATT temp
   FFO test faults at 100degC and clears at 0degC, so any threshold in
   (0, 100) works. *)
astParams_SATT[0].sPmpsState                 := 'AT1K4:L2SI-RTD';
astParams_SATT[0].nRequestAssertionID        := 1100;
astParams_SATT[0].stReactiveParams.nTempSP   := 30;
astParams_SATT[0].stBeamParams.nBeamClass    := 2#0000_0001;
astParams_SATT[0].stBeamParams.neVRange      := 2#1111_1111_1111_1111_1111_1111_1111_1111;
astParams_SATT[0].stBeamParams.nRate         := 10;
astParams_SATT[0].stBeamParams.nTran         := 12;
astParams_SATT[0].stBeamParams.nMachineMode  := 2;

(* ---- SL1L0:POWER (single reactive-temp key; aperture geometry is
   not state-keyed). nTempSP is the RTD fault threshold in degC: the
   SLITS temp FFO test faults at 100degC and clears at 0degC, so any
   threshold in (0, 100) works. *)
astParams_SLITS[0].sPmpsState                := 'SL1L0:POWER-RTD';
astParams_SLITS[0].nRequestAssertionID       := 1200;
astParams_SLITS[0].stReactiveParams.nTempSP  := 30;
astParams_SLITS[0].stBeamParams.nBeamClass   := 2#0000_0001;
astParams_SLITS[0].stBeamParams.neVRange     := 2#1111_1111_1111_1111_1111_1111_1111_1111;
astParams_SLITS[0].stBeamParams.nRate        := 10;
astParams_SLITS[0].stBeamParams.nTran        := 12;
astParams_SLITS[0].stBeamParams.nMachineMode := 2;

(* First helper creates the root document, the rest append. *)
fbJsonHelper_ATM(
    astBeamParams := astParams_ATM,
    bExecute      := TRUE,
    sDevName      := 'TST:ATM',
    bNewDoc       := TRUE);

fbJsonHelper_LIC(
    astBeamParams := astParams_LIC,
    bExecute      := TRUE,
    sDevName      := 'TST:LIC',
    bNewDoc       := FALSE);

fbJsonHelper_PPM(
    astBeamParams := astParams_PPM,
    bExecute      := TRUE,
    sDevName      := 'TST:PPM',
    bNewDoc       := FALSE);

fbJsonHelper_REF(
    astBeamParams := astParams_REF,
    bExecute      := TRUE,
    sDevName      := 'TST:REF',
    bNewDoc       := FALSE);

fbJsonHelper_GBS(
    astBeamParams := astParams_GBS,
    bExecute      := TRUE,
    sDevName      := 'TST:GBS',
    bNewDoc       := FALSE);

fbJsonHelper_IPM(
    astBeamParams := astParams_IPM,
    bExecute      := TRUE,
    sDevName      := 'TST:IPM',
    bNewDoc       := FALSE);

fbJsonHelper_WFS(
    astBeamParams := astParams_WFS,
    bExecute      := TRUE,
    sDevName      := 'TST:WFS',
    bNewDoc       := FALSE);

fbJsonHelper_XPIM(
    astBeamParams := astParams_XPIM,
    bExecute      := TRUE,
    sDevName      := 'TST:XPIM',
    bNewDoc       := FALSE);

fbJsonHelper_SATT(
    astBeamParams := astParams_SATT,
    bExecute      := TRUE,
    sDevName      := 'AT1K4:L2SI',
    bNewDoc       := FALSE);

fbJsonHelper_SLITS(
    astBeamParams := astParams_SLITS,
    bExecute      := TRUE,
    sDevName      := 'SL1L0:POWER',
    bNewDoc       := FALSE);
END_METHOD

END_FUNCTION_BLOCK

// ---- Tests/Helpers/FB_PMPSJsonTestHelper.TcPOU
FUNCTION_BLOCK FB_PMPSJsonTestHelper
(*
    Build a JSON document in memory from the input structs and publish
    it to the global PMPS doc (PMPS_GVL.BP_jsonDoc). Unlike
    FB_PMPSJsonTestHelperEx, this helper serializes the reactive
    temperature and pressure set points (nTempSP / nPressSP) into the
    reactive_temp / reactive_pressure members, so it is the helper to
    use for any device whose test reads a reactive-DB threshold.

    bNewDoc selects the document mode: TRUE creates a fresh root
    document (first device in the seeding chain); FALSE appends this
    device to the existing PMPS_GVL.BP_jsonDoc, so several helpers can
    accumulate into one multi-device document.
*)
VAR_IN_OUT
    astBeamParams: ARRAY[*] OF ST_DbStateParams;
END_VAR
VAR_INPUT
    bExecute: BOOL;
    sDevName: STRING;
    bNewDoc: BOOL;
END_VAR
VAR_OUTPUT
END_VAR
VAR
    rtExec: R_TRIG;
    jsonRoot: SJsonValue;
    jsonDevice: SJsonValue;
    ajsonState: ARRAY[0..GeneralConstants.MAX_STATES] OF SJsonValue;
    fbJson: FB_JsonDomParser;

    nIter: DINT;
    nId: DINT;

    aseVRange: ARRAY[0..GeneralConstants.MAX_STATES] OF STRING;
    asRate: ARRAY[0..GeneralConstants.MAX_STATES] OF STRING;
    asBCRange: ARRAY[0..GeneralConstants.MAX_STATES] OF STRING;
    asTran: ARRAY[0..GeneralConstants.MAX_STATES] OF STRING;

    sTemp: STRING;
    sPress: STRING;
END_VAR


rtExec(CLK:=bExecute);
IF NOT rtExec.Q THEN
    RETURN;
END_IF

IF bNewDoc THEN
    jsonRoot := fbJson.NewDocument();
ELSE
    jsonRoot := PMPS_GVL.BP_jsonDoc;
END_IF
jsonDevice := fbJson.AddObjectMember(jsonRoot, sDevName);
FOR nIter := LOWER_BOUND(astBeamParams, 1) TO UPPER_BOUND(astBeamParams, 1) DO
    ajsonState[nIter] := fbJson.AddObjectMember(jsonDevice, astBeamParams[nIter].sPmpsState);

    // Prefer the seeded assertion ID as the DB 'id' so it is unique and
    // meaningful; fall back to a running counter when a state leaves
    // nRequestAssertionID unset, so 'id' is never 0.
    nId := nId + 1;
    IF astBeamParams[nIter].nRequestAssertionID <> 0 THEN
        fbJson.AddIntMember(
            v:=ajsonState[nIter],
            member:='id',
            value:=UDINT_TO_DINT(astBeamParams[nIter].nRequestAssertionID),
        );
    ELSE
        fbJson.AddIntMember(
            v:=ajsonState[nIter],
            member:='id',
            value:=nId,
        );
    END_IF
    fbJson.AddStringMember(
        v:=ajsonState[nIter],
        member:='beamline',
        value:='tst',
    );
    aseVRange[nIter] := bitmaskToString(astBeamParams[nIter].stBeamParams.neVRange, 32);
    fbJson.AddStringMember(
        v:=ajsonState[nIter],
        member:='neVRange',
        value:=aseVRange[nIter],
    );
    asRate[nIter] := UDINT_TO_STRING(astBeamParams[nIter].stBeamParams.nRate);
    fbJson.AddStringMember(
        v:=ajsonState[nIter],
        member:='nRate',
        value:=asRate[nIter],
    );
    fbJson.AddStringMember(
        v:=ajsonState[nIter],
        member:='ap_ygap',
        value:='',
    );
    fbJson.AddStringMember(
        v:=ajsonState[nIter],
        member:='ap_xgap',
        value:='',
    );
    fbJson.AddStringMember(
        v:=ajsonState[nIter],
        member:='damage_limit',
        value:='',
    );
    fbJson.AddStringMember(
        v:=ajsonState[nIter],
        member:='notes',
        value:='',
    );
    sTemp := TO_STRING(astBeamParams[nIter].stReactiveParams.nTempSP);
    fbJson.AddStringMember(
        v:=ajsonState[nIter],
        member:='reactive_temp',
        value:=sTemp,
    );
    sPress := TO_STRING(astBeamParams[nIter].stReactiveParams.nPressSP);
    fbJson.AddStringMember(
        v:=ajsonState[nIter],
        member:='reactive_pressure',
        value:=sPress,
    );
    asBCRange[nIter] := bitmaskToString(astBeamParams[nIter].stBeamParams.nBCRange, 15);
    fbJson.AddStringMember(
        v:=ajsonState[nIter],
        member:='nBeamClassRange',
        value:=asBCRange[nIter],
    );
    fbJson.AddStringMember(
        v:=ajsonState[nIter],
        member:='name',
        value:=astBeamParams[nIter].sPmpsState,
    );
    asTran[nIter] := REAL_TO_STRING(astBeamParams[nIter].stBeamParams.nTran);
    fbJson.AddStringMember(
        v:=ajsonState[nIter],
        member:='nTran',
        value:=asTran[nIter],
    );
    fbJson.AddStringMember(
        v:=ajsonState[nIter],
        member:='ap_name',
        value:='None',
    );
    fbJson.AddStringMember(
        v:=ajsonState[nIter],
        member:='ap_ycenter',
        value:='',
    );
    fbJson.AddStringMember(
        v:=ajsonState[nIter],
        member:='ap_xcenter',
        value:='',
    );
    fbJson.AddStringMember(
        v:=ajsonState[nIter],
        member:='pulse_energy',
        value:='',
    );
    fbJson.AddBoolMember(
        v:=ajsonState[nIter],
        member:='special',
        value:=FALSE,
    );
END_FOR

PMPS_GVL.BP_jsonDoc := jsonRoot;

METHOD bitmaskToString : STRING
VAR_INPUT
    nBitmask: DWORD;
    nBits: UINT;
END_VAR
VAR
    nIter: UINT;
END_VAR

bitmaskToString := '';
FOR nIter := 1 TO nBits DO
    bitmaskToString := CONCAT(DWORD_TO_STRING(SHR(nBitmask, nIter - 1) AND 1), bitmaskToString);
END_FOR
END_METHOD

END_FUNCTION_BLOCK

// ---- Tests/FB_ATMTest.TcPOU
FUNCTION_BLOCK FB_ATMTest EXTENDS FB_TestSuite
VAR
    (* Caller-owned axis, persistent storage, and Y motor.
       In a real PRG the AxisRef would come from MAIN.Mxx. *)
    axRef    : ARRAY[1..2] OF AXIS_REF;
    fbPDS    : LCLS_Tc_DevAbs.FB_PersistentDataStorage;
    // X motor (align target to beam)
    fbMotorX : FB_MotionStageNC(AxisRef := axRef[1], iPersistentDataStorage := fbPDS, sName := 'X');
    (* FB_ATM is single-axis (nActiveMotorCount := 1), so only slot 1
       holds a real motor. aiMotionStage is sized to
       MotionConstants.MAX_STATE_MOTORS to match FB_ATM.FB_Init's
       fixed-size signature; slots 2-4 default-init to a nil interface
       and are never touched. *)
    fbMotorY : FB_MotionStageNC(AxisRef := axRef[2], iPersistentDataStorage := fbPDS, sName := 'Y');
    aiMotionStage : ARRAY[1..MotionConstants.MAX_STATE_MOTORS] OF I_MotionStage := [fbMotorY];

    {attribute 'pytmc' := '
        pv: MMS
        array: 1..1 | 1..6
    '}
    astPositionState : ARRAY[1..MotionConstants.MAX_STATE_MOTORS]
                         OF ARRAY[1..GeneralConstants.MAX_STATES] OF ST_PositionState;

    fbFFHWO    : FB_HardwareFFOutput;
    fbArbiter  : FB_Arbiter(1);
    fbSubSysIO : FB_DummyArbIO;

    sDeviceName    : STRING := 'TST:ATM';
    sTransitionKey : STRING := 'TST:ATM-TRANSITION';

    (* Caller-owned file-reader status, bound to FB_ATM by REFERENCE
       TO. In a real PRG these point at MOTION_GVL.fbPmpsFileReader;
       here they stay FALSE so the DB read proceeds. *)
    bFileReaderBusy  : BOOL;
    bFileReaderError : BOOL;

    fbATM : FB_ATM(
        aiMotionStage         := aiMotionStage,
        astPositionState      := astPositionState,
        fbFFHWO               := fbFFHWO,
        fbArbiter             := fbArbiter,
        sDeviceName           := sDeviceName,
        sTransitionKey        := sTransitionKey,
        bEnableBeamParams     := TRUE,
        bEnablePositionLimits := TRUE,
        bReadDBNow            := TRUE,
        bFileReaderBusy       := bFileReaderBusy,
        bFileReaderError      := bFileReaderError
    );

    (* stDefault is the caller-owned
       baseline template that FB_CC_StatePMPSConfig's inner FB_StateSetup
       preloads from; fbATM subsequently overrides per-state sName and
       fDelta via its own FB_CC_InternalStateConfig array. *)
    stDefault : ST_PositionState := (
        bMoveOk       := TRUE,
        bValid        := TRUE,
        bUseRawCounts := FALSE
    );

    afbStatePMPS : ARRAY[1..6] OF FB_CC_StatePMPSConfig[
        (stPositionState := astPositionState[1][E_ATM_States.OUT],
         stDefault       := stDefault,
         fPosition       := 10,
         sPmpsState      := 'TST:ATM-OUT'),
        (stPositionState := astPositionState[1][E_ATM_States.TARGET1],
         stDefault       := stDefault,
         fPosition       := 20,
         sPmpsState      := 'TST:ATM-TARGET1'),
        (stPositionState := astPositionState[1][E_ATM_States.TARGET2],
         stDefault       := stDefault,
         fPosition       := 30,
         sPmpsState      := 'TST:ATM-TARGET2'),
        (stPositionState := astPositionState[1][E_ATM_States.TARGET3],
         stDefault       := stDefault,
         fPosition       := 40,
         sPmpsState      := 'TST:ATM-TARGET3'),
        (stPositionState := astPositionState[1][E_ATM_States.TARGET4],
         stDefault       := stDefault,
         fPosition       := 50,
         sPmpsState      := 'TST:ATM-TARGET4'),
        (stPositionState := astPositionState[1][E_ATM_States.TARGET5],
         stDefault       := stDefault,
         fPosition       := 60,
         sPmpsState      := 'TST:ATM-TARGET5')
    ];

    bFirstScan : BOOL := TRUE;
    i          : UINT;
END_VAR

IF bFirstScan THEN
    fbMotorY.SetModeEnableLimits(
        LimBackward    := TRUE,
        LimForward     := TRUE,
        HomeEnable     := FALSE,
        BrakeMode      := E_StageBrakeMode.IF_ENABLED,
        EnableMode     := E_StageEnableMode.DURING_MOTION,
        HomeMode       := E_EpicsHomeCmd.LOW_LIMIT,
        UserEnable     := TRUE,
        HardwareEnable := TRUE
    );
    fbMotorX.SetModeEnableLimits(
        LimBackward    := TRUE,
        LimForward     := TRUE,
        HomeEnable     := FALSE,
        BrakeMode      := E_StageBrakeMode.IF_ENABLED,
        EnableMode     := E_StageEnableMode.DURING_MOTION,
        HomeMode       := E_EpicsHomeCmd.LOW_LIMIT,
        UserEnable     := TRUE,
        HardwareEnable := TRUE
    );
    fbMotorX.SetVelocity(Velocity := 15.5);
    fbMotorX.RestoreMotionParams      := FALSE;
    fbMotorX.DoNotRestoreNcParameters := TRUE;
    fbMotorY.SetVelocity(Velocity := 15.5);
    fbMotorY.RestoreMotionParams      := FALSE;
    fbMotorY.DoNotRestoreNcParameters := TRUE;
    bFileReaderBusy  := TRUE;
    bFileReaderError := FALSE;
    bFirstScan := FALSE;
END_IF

TestStateMove();
TestTempFFO();

(* Fake PMPS handling. *)
fbSubSysIO(
    LA  := fbArbiter,
    FFO := fbFFHWO
);
fbPDS();
fbMotorX();
fbMotorY();
fbATM();

bFileReaderBusy  := FALSE;
bFileReaderError := FALSE;

METHOD SetATMTemp
VAR_INPUT
    iTempC : INT;
END_VAR
VAR
    ptr : POINTER TO INT;
END_VAR
ptr  := ADR(fbATM.fbTempSensor1.iRaw);
ptr^ := iTempC * 10;
END_METHOD

(*
    Smoke test for ATM state-move wiring. Walks OUT then TARGET1 and
    asserts each lands within fTolerance of the configured fPosition.
    Mirrors FB_REFTest: stageReady gate up front, NOT bMoving +
    position-tolerance check per state, 60s watchdog, on timeout
    AssertTrue(FALSE, ...) with the current step and observed
    position. Two moves is enough to exercise the FB wiring; the
    motion stack itself is covered by the
    lcls-twincat-motion-abstraction test suite.
*)
METHOD TestStateMove
VAR_INST
    tonTimer  : TON;
    nTestStep : INT := 0;
    fObserved : LREAL;
END_VAR
VAR CONSTANT
    fTolerance : LREAL := 2.0;
END_VAR
TEST('TestATMStateMove');


tonTimer(IN := TRUE, PT := T#60s);
fObserved := fbMotorY.stMotionStatus.fActPosition;

CASE nTestStep OF
    0:
        IF fbMotorY.stMotionStatus.bStageReady
           AND NOT fbMotorY.stMotionStatus.bError THEN
            fbATM.eEnumSet := E_ATM_States.OUT;
            nTestStep      := 1;
        END_IF
    1:
        (* OUT is configured at fPosition := 10 in afbStatePMPS[1]. *)
        IF fbATM.eEnumGet = E_ATM_States.OUT
           AND NOT fbMotorY.stMotionStatus.bMoving
           AND ABS(fObserved - 10.0) <= fTolerance THEN
            fbATM.eEnumSet := E_ATM_States.TARGET1;
            nTestStep      := 2;
        END_IF
    2:
        (* TARGET1 is configured at fPosition := 20 in afbStatePMPS[2]. *)
        IF fbATM.eEnumGet = E_ATM_States.TARGET1
           AND NOT fbMotorY.stMotionStatus.bMoving
           AND ABS(fObserved - 20.0) <= fTolerance THEN
            AssertTrue(
                Condition := TRUE,
                Message   := 'TestATMStateMove: OUT then TARGET1 reached within tolerance');
            nTestStep := 3;
        END_IF
END_CASE

IF nTestStep = 3 THEN
    TEST_FINISHED();
ELSIF tonTimer.Q THEN
    AssertTrue(
        Condition := FALSE,
        Message   := CONCAT(
            CONCAT(
                CONCAT('TestATMStateMove: timed out at step ', TO_STRING(nTestStep)),
                CONCAT(', eEnumGet=', TO_STRING(TO_UDINT(fbATM.eEnumGet)))),
            CONCAT(', fActPos=', TO_STRING(fObserved))));
    TEST_FINISHED();
END_IF
END_METHOD

METHOD TestTempFFO
VAR_INST
    tonTimer    : TON;
    nStep       : UINT := 0;
    bOutChecked : BOOL := FALSE;
    bInChecked  : BOOL := FALSE;
END_VAR
VAR CONSTANT
    nLastStep : UINT := 3;
END_VAR

(* Do we fault at the correct times?
   Parasitically depends on state move test. *)
TEST('TestATMTempFFO');

(* Prepare a timeout *)
tonTimer(IN := TRUE, PT := T#10s);

CASE nStep OF
    0:
        (* Set the thermocouple temperature to crazy high number. *)
        SetATMTemp(100);
        nStep := nStep + 1;
    1:
        (* Wait till we see "OUT" state and one other state (OUT
           should be no fault). *)
        IF fbATM.eEnumGet = E_ATM_States.OUT THEN
            AssertTrue(
                fbATM.fbTempSensor1.FFO.i_xOK,
                'Faulted even in out position!'
            );
            bOutChecked := TRUE;
        ELSIF fbATM.eEnumGet <> E_ATM_States.Unknown THEN
            AssertFalse(
                fbATM.fbTempSensor1.FFO.i_xOK,
                'No fault even for an in position!'
            );
            bInChecked := TRUE;
        END_IF
        IF bOutChecked AND bInChecked THEN
            nStep := nStep + 1;
        END_IF
    2:
        (* Set the thermocouple temperature to low again. *)
        SetATMTemp(0);
        nStep := nStep + 1;
    3:
        AssertTrue(
            fbATM.fbTempSensor1.FFO.i_xOK,
            'Faulted even with low temp!'
        );
        nStep := nStep + 1;
END_CASE

IF tonTimer.Q OR nStep > nLastStep THEN
    AssertFalse(tonTimer.Q, 'Timeout in ATM temp FFO test');
    TEST_FINISHED();
END_IF
END_METHOD

END_FUNCTION_BLOCK

// ---- Devices/ATM/FB_ATM.TcPOU
(* Arrival Time Monitor (ATM): thin ND-framework state-mover wrapper.
   Y mover via FB_PositionStatePMPSND (states OUT, TARGET1..TARGET5),
   plus a tick site for the in-beam thermocouple and flow meter.
   Caller-owned deps injected via FB_Init REFERENCE TO and forwarded to
   fbStates; device enum bridge and toggles re-forwarded each cycle. *)
{attribute 'call_after_init'}
FUNCTION_BLOCK FB_ATM
VAR_INPUT
    (* Device-specific state-enum bridges. Typed as E_ATM_States (UINT
       base) so the caller surface is enum-checked; the inline-init
       below binds them to FB_PositionStatePMPSND's REFERENCE TO UINT
       params via the shared UINT base. Callers drive moves with
       `fbATM.eEnumSet := E_ATM_States.TARGET1;` and read
       `fbATM.eEnumGet`. *)
    // Set this to a non-unknown value to request a new move.
    {attribute 'pytmc' := '
        pv: MMS:STATE:SET
        io: io
    '}
    eEnumSet : E_ATM_States;
END_VAR
VAR

    {attribute 'pytmc' := 'pv: STC:01'}
    fbTempSensor1 : FB_CC_TempSensor;

    {attribute 'pytmc' := 'pv: FWM'}
    fbFlowMeter : FB_AnalogInput := (iTermBits := 15, fTermMax := 60, fTermMin := 0);

    (* REFERENCE TO backing fields populated by FB_Init. Same names as
       FB_Init params; THIS^. disambiguates inside FB_Init.
       Live-bound to caller storage for the lifetime of the FB. *)
    {attribute 'no_copy'}
    aiMotionStage         : REFERENCE TO ARRAY[1..MotionConstants.MAX_STATE_MOTORS] OF I_MotionStage;
    {attribute 'no_copy'}
    astPositionState      : REFERENCE TO ARRAY[1..MotionConstants.MAX_STATE_MOTORS]
                                            OF ARRAY[1..GeneralConstants.MAX_STATES] OF ST_PositionState;
    {attribute 'no_copy'}
    fbFFHWO               : REFERENCE TO FB_HardwareFFOutput;
    {attribute 'no_copy'}
    fbArbiter             : REFERENCE TO FB_Arbiter;
    sDeviceName           : STRING;
    sTransitionKey        : STRING;
    bEnableMotion         : BOOL := TRUE;
    bEnableBeamParams     : BOOL;
    bEnablePositionLimits : BOOL;
    bReadDBNow            : BOOL;
    bFileReaderBusy       : REFERENCE TO BOOL;
    bFileReaderError      : REFERENCE TO BOOL;

    (* One configurator per ATM state (OUT + 5 targets). Writes the
       per-state sName and fDelta. Ticked cyclically in the body AFTER
       fbStates so its writes win over the template baseline
       FB_StateSetup applied via FB_CC_StatePMPSConfig. Idempotent once
       stPositionState.bUpdated trips. *)
    afbStateDefaults : ARRAY[1..6] OF FB_CC_InternalStateConfig[
        (stPositionState := astPositionState[1][E_ATM_States.OUT],
         sName           := 'OUT',
         fDelta          := FDELTA_DEFAULT),
        (stPositionState := astPositionState[1][E_ATM_States.TARGET1],
         sName           := 'TARGET1',
         fDelta          := FDELTA_DEFAULT),
        (stPositionState := astPositionState[1][E_ATM_States.TARGET2],
         sName           := 'TARGET2',
         fDelta          := FDELTA_DEFAULT),
        (stPositionState := astPositionState[1][E_ATM_States.TARGET3],
         sName           := 'TARGET3',
         fDelta          := FDELTA_DEFAULT),
        (stPositionState := astPositionState[1][E_ATM_States.TARGET4],
         sName           := 'TARGET4',
         fDelta          := FDELTA_DEFAULT),
        (stPositionState := astPositionState[1][E_ATM_States.TARGET5],
         sName           := 'TARGET5',
         fDelta          := FDELTA_DEFAULT)
    ];

    {attribute 'pytmc' := 'pv: MMS'}
    fbStates : FB_PositionStatePMPSND(
        aiMotionStage         := aiMotionStage,
        astPositionState      := astPositionState,
        nActiveMotorCount     := 1,
        eEnumSet              := eEnumSet,
        eEnumGet              := eEnumGet,
        bEnableMotion         := bEnableMotion,
        eMotionRequestPolicy  := E_MotionRequestPolicy.INTERRUPT,
        bEnableBeamParams     := bEnableBeamParams,
        bEnablePositionLimits := bEnablePositionLimits,
        bReadDBNow            := bReadDBNow,
        bFileReaderBusy       := bFileReaderBusy,
        bFileReaderError      := bFileReaderError,
        fbFFHWO               := fbFFHWO,
        fbArbiter             := fbArbiter,
        sDeviceName           := sDeviceName,
        sTransitionKey        := sTransitionKey
    );
    i : UINT;
END_VAR
VAR_OUTPUT
    // The current position state as an enum.
    {attribute 'pytmc' := '
        pv: MMS:STATE:GET
        io: i
    '}
    eEnumGet: E_ATM_States;
    // The PMPS database lookup associated with the current position state.
    stDbStateParams: ST_DbStateParams;
END_VAR
VAR CONSTANT
    (* ATM-wide default tolerance for state in-position detection,
       applied per-state by afbStateDefaults. *)
    FDELTA_DEFAULT : LREAL := 2;
END_VAR

IF NOT __ISVALIDREF(aiMotionStage)
   OR NOT __ISVALIDREF(astPositionState)
   OR NOT __ISVALIDREF(fbFFHWO)
   OR NOT __ISVALIDREF(fbArbiter) THEN
    RETURN;
END_IF

(* Device-side per-state defaults (afbStateDefaults) are written
   once in FB_CC_InternalStateConfig.CallAfterInit; no cyclic tick. *)
fbStates(stDbStateParams=> stDbStateParams);

(* In-beam thermocouple: only faults when something is actually in the
   beam (i.e. not OUT). Driven by the PMPS DB temp setpoint. *)
fbTempSensor1(
    fFaultThreshold := fbStates.stDbStateParams.stReactiveParams.nTempSP,
    bVeto           := eEnumGet = E_ATM_States.OUT,
    sDevName        := sDeviceName,
    io_fbFFHWO      := fbFFHWO
);

fbFlowMeter();

(* Auto-fired after FB_Init. fbStates' inline-init ran first and
   forwarded nil refs, so this re-supplies the now-valid refs via
   fbStates.CallAfterInitStateMover / CallAfterInitPMPS and writes the
   per-state device defaults. *)
{attribute 'call_after_init'}
METHOD CallAfterInit
afbStateDefaults[1].CallAfterInit(stPositionState := THIS^.astPositionState[1][E_ATM_States.OUT]);
afbStateDefaults[2].CallAfterInit(stPositionState := THIS^.astPositionState[1][E_ATM_States.TARGET1]);
afbStateDefaults[3].CallAfterInit(stPositionState := THIS^.astPositionState[1][E_ATM_States.TARGET2]);
afbStateDefaults[4].CallAfterInit(stPositionState := THIS^.astPositionState[1][E_ATM_States.TARGET3]);
afbStateDefaults[5].CallAfterInit(stPositionState := THIS^.astPositionState[1][E_ATM_States.TARGET4]);
afbStateDefaults[6].CallAfterInit(stPositionState := THIS^.astPositionState[1][E_ATM_States.TARGET5]);

THIS^.fbStates.CallAfterInitStateMover(
    aiMotionStage         := aiMotionStage,
    astPositionState      := astPositionState,
    nActiveMotorCount     := 1,
    eEnumSet              := eEnumSet,
    eEnumGet              := eEnumGet,
    bEnableMotion         := bEnableMotion,
    eMotionRequestPolicy  := E_MotionRequestPolicy.INTERRUPT,
);

THIS^.fbStates.CallAfterInitPMPS(
    aiMotionStage         := aiMotionStage,
    astPositionState      := astPositionState,
    bEnableBeamParams     := bEnableBeamParams,
    bEnablePositionLimits := bEnablePositionLimits,
    bReadDBNow            := bReadDBNow,
    bFileReaderBusy       := bFileReaderBusy,
    bFileReaderError      := bFileReaderError,
    fbFFHWO               := fbFFHWO,
    fbArbiter             := fbArbiter,
    sDeviceName           := sDeviceName,
    sTransitionKey        := sTransitionKey
);
END_METHOD

(* Stores FB_Init inputs into instance fields; every non-value input is
   REFERENCE TO, REF= bound for the FB lifetime. fbStates inline-init
   captured these params at construction, so this records the same refs
   on THIS^ for body use and live caller writes. *)
{attribute 'analysis' := '-33'}
METHOD FB_Init : BOOL
VAR_INPUT
    bInitRetains           : BOOL;
    bInCopyCode            : BOOL;
    aiMotionStage          : REFERENCE TO ARRAY[1..MotionConstants.MAX_STATE_MOTORS] OF I_MotionStage;
    astPositionState       : REFERENCE TO ARRAY[1..MotionConstants.MAX_STATE_MOTORS]
                                            OF ARRAY[1..GeneralConstants.MAX_STATES] OF ST_PositionState;
    fbFFHWO                : REFERENCE TO FB_HardwareFFOutput;
    fbArbiter              : REFERENCE TO FB_Arbiter;
    sDeviceName            : STRING;
    sTransitionKey         : STRING;
    bEnableBeamParams      : BOOL;
    bEnablePositionLimits  : BOOL;
    bReadDBNow             : BOOL;
    bFileReaderBusy       : REFERENCE TO BOOL;
    bFileReaderError      : REFERENCE TO BOOL;
END_VAR
THIS^.aiMotionStage    REF= aiMotionStage;
THIS^.astPositionState REF= astPositionState;
THIS^.fbFFHWO          REF= fbFFHWO;
THIS^.fbArbiter        REF= fbArbiter;
THIS^.sDeviceName      := sDeviceName;
THIS^.sTransitionKey   := sTransitionKey;
THIS^.bEnableBeamParams     := bEnableBeamParams;
THIS^.bEnablePositionLimits := bEnablePositionLimits;
THIS^.bReadDBNow            := bReadDBNow;
THIS^.bFileReaderBusy       REF= bFileReaderBusy;
THIS^.bFileReaderError      REF= bFileReaderError;
END_METHOD

END_FUNCTION_BLOCK

// ---- POUs/FB_CC_TempSensor.TcPOU
FUNCTION_BLOCK FB_CC_TempSensor EXTENDS FB_TempSensor_FFO
VAR
    rtVetoReset: R_TRIG;
END_VAR

// Reset the FFO for transitions to bVeto
// bAutoreset is False, but we still want to clear the fault on veto
rtVetoReset(CLK:=bVeto);
FFO.i_xReset := rtVetoReset.Q;

SUPER^(bAutoReset:=FALSE, io_fbFFHWO:=io_fbFFHWO);

END_FUNCTION_BLOCK

// ---- POUs/FB_CC_InternalStateConfig.TcPOU
(*
    Per-(state) writer of the device-FB-side fields of an
    ST_PositionState slot that FB_CC_StatePMPSConfig does not
    touch. Performs a one-shot direct write of sName (per-state
    label) and fDelta (per-state tolerance) from CallAfterInit.
    Owned by the device FB (e.g. FB_ATM), one instance per state,
    both fields hardcoded inside the device FB.

    Other slot fields (fPosition, sPmpsState, and the
    safety/baseline fields) are owned by FB_CC_StatePMPSConfig on
    the integrator side; the two helpers' writes do not overlap so
    their CallAfterInit ordering is irrelevant.

    The FB body is empty; the slot is never touched cyclically, so
    online-view edits persist.
*)
FUNCTION_BLOCK FB_CC_InternalStateConfig
VAR_INPUT
END_VAR
VAR
    {attribute 'no_copy'}
    stPositionState : REFERENCE TO ST_PositionState;
    sName           : STRING;
    fDelta          : LREAL;
END_VAR

(* One-shot write of the device-owned per-state fields (sName,
   fDelta) into the slot. *)
METHOD CallAfterInit
VAR_INPUT
    stPositionState : REFERENCE TO ST_PositionState;
END_VAR
THIS^.stPositionState REF= stPositionState;

IF __ISVALIDREF(THIS^.stPositionState) THEN
    THIS^.stPositionState.sName  := THIS^.sName;
    THIS^.stPositionState.fDelta := THIS^.fDelta;
END_IF
END_METHOD

(* Stores the slot reference plus the per-state sName and fDelta
   at instantiation. *)
METHOD FB_Init : BOOL
VAR_INPUT
    bInitRetains    : BOOL;
    bInCopyCode     : BOOL;
    stPositionState : REFERENCE TO ST_PositionState;
    sName           : STRING;
    fDelta          : LREAL;
END_VAR
THIS^.stPositionState REF= stPositionState;
THIS^.sName            := sName;
THIS^.fDelta           := fDelta;
END_METHOD

END_FUNCTION_BLOCK

// ---- POUs/FB_CC_StatePMPSConfig.TcPOU
(*
    Per-(state) writer of an ST_PositionState slot. Owned by the
    integrator PRG. Stripped-down counterpart of motion-lib's
    FB_PMPSStateConfigurator.

    Performs a one-shot direct write of the slot from CallAfterInit:
    copies the caller's stDefault baseline for the safety-relevant
    fields (bMoveOk, bValid, bUseRawCounts, bLocked, nEncoderCount),
    then overlays fPosition and stPMPS.sPmpsState. sName and fDelta
    are deliberately NOT touched here: they are owned by the device
    FB's FB_CC_InternalStateConfig array, so the two helpers' writes
    do not overlap and their CallAfterInit ordering is irrelevant.

    The FB body is empty; the inner FB_StateSetup is wired (refs +
    template preload) at init purely as a defensive backstop, so that
    a stray cyclic call to fbStateSetup stays safe and template-aware.

    Online-view edits to the slot persist because nothing writes it
    after init.
*)
{attribute 'call_after_init'}
FUNCTION_BLOCK FB_CC_StatePMPSConfig
VAR_INPUT
END_VAR
VAR
    {attribute 'no_copy'}
    stPositionState : REFERENCE TO ST_PositionState;
    {attribute 'no_copy'}
    stDefault       : REFERENCE TO ST_PositionState;
    fPosition       : LREAL;
    sPmpsState      : STRING;
    fbStateSetup    : FB_StateSetup(
        stDefault       := stDefault,
        stPositionState := stPositionState,
        bSetDefault     := TRUE
    );
END_VAR

(* Re-binds the inner FB_StateSetup's REFs after FB_Init (defensive),
   then performs a one-shot write of the slot: safety/baseline fields
   from stDefault and fPosition / sPmpsState overlay. sName and fDelta
   are owned by FB_CC_InternalStateConfig. *)
{attribute 'call_after_init'}
METHOD CallAfterInit
VAR_INPUT
END_VAR
THIS^.fbStateSetup.CallAfterInit(
    stDefault       := THIS^.stDefault,
    stPositionState := THIS^.stPositionState,
    bSetDefault     := TRUE
);

IF __ISVALIDREF(THIS^.stPositionState) AND __ISVALIDREF(THIS^.stDefault) THEN
    THIS^.stPositionState.bMoveOk       := THIS^.stDefault.bMoveOk;
    THIS^.stPositionState.bValid        := THIS^.stDefault.bValid;
    THIS^.stPositionState.bUseRawCounts := THIS^.stDefault.bUseRawCounts;
    THIS^.stPositionState.bLocked       := THIS^.stDefault.bLocked;
    THIS^.stPositionState.nEncoderCount := THIS^.stDefault.nEncoderCount;

    THIS^.stPositionState.fPosition         := THIS^.fPosition;
    THIS^.stPositionState.stPMPS.sPmpsState := THIS^.sPmpsState;
END_IF
END_METHOD

(* Stores the slot reference, the device-common stDefault template
   REF, plus the per-install fPosition + sPmpsState at instantiation. *)
METHOD FB_Init : BOOL
VAR_INPUT
    bInitRetains    : BOOL;
    bInCopyCode     : BOOL;
    stPositionState : REFERENCE TO ST_PositionState;
    stDefault       : REFERENCE TO ST_PositionState;
    fPosition       : LREAL;
    sPmpsState      : STRING;
END_VAR
THIS^.stPositionState REF= stPositionState;
THIS^.stDefault       REF= stDefault;
THIS^.fPosition        := fPosition;
THIS^.sPmpsState       := sPmpsState;
END_METHOD

END_FUNCTION_BLOCK

// ---- Tests/FB_GBSTest.TcPOU
(* Integration smoke for FB_GBS. TestStateMove proves the wrapper wiring
   (REFERENCE TO refs, CallAfterInit chain, fbStates inline-init, per-state
   defaults, PMPS key registration) drives the motor to the configured
   fPosition for OUT then TARGET1a. TestTempFFO proves the two in-beam RTDs
   fault only in a target state, vetoed while OUT. Motion stack tested elsewhere. *)
{attribute 'analysis' := '-33'}
FUNCTION_BLOCK FB_GBSTest EXTENDS FB_TestSuite
VAR
    (* Caller-owned axis, persistent storage, and Y motor.
       In a real PRG the AxisRef would come from MAIN.Mxx. *)
    axRef    : AXIS_REF;
    fbPDS    : LCLS_Tc_DevAbs.FB_PersistentDataStorage;

    (* FB_GBS is single-axis (nActiveMotorCount := 1), so only slot 1
       holds a real motor. aiMotionStage is sized to
       MotionConstants.MAX_STATE_MOTORS to match FB_GBS.FB_Init's
       fixed-size signature; slots 2-4 default-init to a nil interface
       and are never touched. *)
    fbMotorY : FB_MotionStageNC(AxisRef := axRef, iPersistentDataStorage := fbPDS, sName := 'Y');
    aiMotionStage : ARRAY[1..MotionConstants.MAX_STATE_MOTORS] OF I_MotionStage := [fbMotorY];

    {attribute 'pytmc' := '
        pv: MMS
        array: 1..1 | 1..4
    '}
    astPositionState : ARRAY[1..MotionConstants.MAX_STATE_MOTORS]
                         OF ARRAY[1..GeneralConstants.MAX_STATES] OF ST_PositionState;

    fbFFHWO    : FB_HardwareFFOutput;
    fbArbiter  : FB_Arbiter(1);
    fbSubSysIO : FB_DummyArbIO;

    sDeviceName    : STRING := 'TST:GBS';
    sTransitionKey : STRING := 'TST:GBS-TRANSITION';

    (* Caller-owned file-reader status, bound to FB_GBS by REFERENCE
       TO. In a real PRG these point at MOTION_GVL.fbPmpsFileReader;
       here they stay FALSE so the DB read proceeds. *)
    bFileReaderBusy  : BOOL;
    bFileReaderError : BOOL;

    fbGBS : FB_GBS(
        aiMotionStage         := aiMotionStage,
        astPositionState      := astPositionState,
        fbFFHWO               := fbFFHWO,
        fbArbiter             := fbArbiter,
        sDeviceName           := sDeviceName,
        sTransitionKey        := sTransitionKey,
        bEnableBeamParams     := TRUE,
        bEnablePositionLimits := TRUE,
        bReadDBNow            := TRUE,
        bFileReaderBusy       := bFileReaderBusy,
        bFileReaderError      := bFileReaderError
    );

    (* Per-install PMPS-side state config (caller-owned). Mirrors what
       a real PRG_xxL0_GBS would declare. stDefault is the caller-owned
       baseline template that FB_CC_StatePMPSConfig's inner FB_StateSetup
       preloads from; fbGBS subsequently overrides per-state sName and
       fDelta via its own FB_CC_InternalStateConfig array. sPmpsState
       keys match the fake DB seeded by FB_CC_PMPSTestSetup. *)
    stDefault : ST_PositionState := (
        bMoveOk       := TRUE,
        bValid        := TRUE,
        bUseRawCounts := FALSE
    );

    afbStatePMPS : ARRAY[1..10] OF FB_CC_StatePMPSConfig[
        (stPositionState := astPositionState[1][E_GBS_States.OUT],
         stDefault       := stDefault,
         fPosition       := 10,
         sPmpsState      := 'TST:GBS-OUT'),
        (stPositionState := astPositionState[1][E_GBS_States.TARGET1a],
         stDefault       := stDefault,
         fPosition       := 20,
         sPmpsState      := 'TST:GBS-TARGET1a'),
        (stPositionState := astPositionState[1][E_GBS_States.TARGET1b],
         stDefault       := stDefault,
         fPosition       := 30,
         sPmpsState      := 'TST:GBS-TARGET1b'),
        (stPositionState := astPositionState[1][E_GBS_States.TARGET2a],
         stDefault       := stDefault,
         fPosition       := 40,
         sPmpsState      := 'TST:GBS-TARGET2a'),
        (stPositionState := astPositionState[1][E_GBS_States.TARGET2b],
         stDefault       := stDefault,
         fPosition       := 50,
         sPmpsState      := 'TST:GBS-TARGET2b'),
        (stPositionState := astPositionState[1][E_GBS_States.TARGET3a],
         stDefault       := stDefault,
         fPosition       := 60,
         sPmpsState      := 'TST:GBS-TARGET3a'),
        (stPositionState := astPositionState[1][E_GBS_States.TARGET3b],
         stDefault       := stDefault,
         fPosition       := 70,
         sPmpsState      := 'TST:GBS-TARGET3b'),
        (stPositionState := astPositionState[1][E_GBS_States.TARGET4],
         stDefault       := stDefault,
         fPosition       := 80,
         sPmpsState      := 'TST:GBS-TARGET4'),
        (stPositionState := astPositionState[1][E_GBS_States.TARGET5],
         stDefault       := stDefault,
         fPosition       := 90,
         sPmpsState      := 'TST:GBS-TARGET5'),
        (stPositionState := astPositionState[1][E_GBS_States.TARGET6],
         stDefault       := stDefault,
         fPosition       := 100,
         sPmpsState      := 'TST:GBS-TARGET6')
    ];

    bFirstScan : BOOL := TRUE;
    i          : UINT;
END_VAR

TestStateMove();
TestTempFFO();

METHOD AssertBothTempFault
VAR_INPUT
    Message : STRING;
END_VAR
AssertFalse(
    fbGBS.fbRTD1.FFO.i_xOK,
    CONCAT('GBS RTD1 expected fault: ', Message)
);
AssertFalse(
    fbGBS.fbRTD2.FFO.i_xOK,
    CONCAT('GBS RTD2 expected fault: ', Message)
);
END_METHOD

METHOD AssertNeitherTempFault
VAR_INPUT
    Message : STRING;
END_VAR
AssertTrue(
    fbGBS.fbRTD1.FFO.i_xOK,
    CONCAT('GBS RTD1 expected ok: ', Message)
);
AssertTrue(
    fbGBS.fbRTD2.FFO.i_xOK,
    CONCAT('GBS RTD2 expected ok: ', Message)
);
END_METHOD

METHOD SetGBSTemp
VAR_INPUT
    iTempC : INT;
END_VAR
VAR
    ptr : POINTER TO INT;
END_VAR
ptr  := ADR(fbGBS.fbRTD1.iRaw);
ptr^ := iTempC * 10;

ptr  := ADR(fbGBS.fbRTD2.iRaw);
ptr^ := iTempC * 10;
END_METHOD

(* Smoke test for GBS state-move wiring. Walks OUT then TARGET1a and asserts
   each lands within fTolerance of the configured fPosition. Mirrors FB_PPMTest:
   stageReady gate, NOT bMoving + tolerance check per state, 60s watchdog, on
   timeout AssertTrue(FALSE, ...) with the step and observed position. *)
METHOD TestStateMove
VAR_INST
    tonTimer  : TON;
    nTestStep : INT := 0;
    fObserved : LREAL;
END_VAR
VAR CONSTANT
    fTolerance : LREAL := 2.0;
END_VAR
TEST('TestGBSStateMove');

tonTimer(IN := TRUE, PT := T#60s);
fObserved := fbMotorY.stMotionStatus.fActPosition;

CASE nTestStep OF
    0:
        IF bFirstScan THEN
            fbMotorY.SetModeEnableLimits(
                LimBackward    := TRUE,
                LimForward     := TRUE,
                HomeEnable     := FALSE,
                BrakeMode      := E_StageBrakeMode.IF_ENABLED,
                EnableMode     := E_StageEnableMode.DURING_MOTION,
                HomeMode       := E_EpicsHomeCmd.LOW_LIMIT,
                UserEnable     := TRUE,
                HardwareEnable := TRUE
            );
            fbMotorY.SetVelocity(Velocity := 15.5);
            fbMotorY.RestoreMotionParams      := FALSE;
            fbMotorY.DoNotRestoreNcParameters := TRUE;
            bFileReaderBusy  := TRUE;
            bFileReaderError := FALSE;
            bFirstScan := FALSE;
        END_IF
        nTestStep      := 1;
    1:
        IF fbMotorY.stMotionStatus.bStageReady
           AND NOT fbMotorY.stMotionStatus.bError THEN
            fbGBS.eEnumSet := E_GBS_States.OUT;
            nTestStep      := 2;
        END_IF
    2:
        (* OUT is configured at fPosition := 10 in afbStatePMPS[1]. *)
        IF fbGBS.eEnumGet = E_GBS_States.OUT
           AND NOT fbMotorY.stMotionStatus.bMoving
           AND ABS(fObserved - 10.0) <= fTolerance THEN
            fbGBS.eEnumSet := E_GBS_States.TARGET1a;
            nTestStep      := 3;
        END_IF
    3:
        (* TARGET1a is configured at fPosition := 20 in afbStatePMPS[2]. *)
        IF fbGBS.eEnumGet = E_GBS_States.TARGET1a
           AND NOT fbMotorY.stMotionStatus.bMoving
           AND ABS(fObserved - 20.0) <= fTolerance THEN
            AssertTrue(
                Condition := TRUE,
                Message   := 'TestGBSStateMove: OUT then TARGET1a reached within tolerance');
            nTestStep := 4;
        END_IF
END_CASE

(* Fake PMPS handling. *)
fbSubSysIO(
    LA  := fbArbiter,
    FFO := fbFFHWO
);

fbPDS();
fbMotorY();
fbGBS();

bFileReaderBusy  := FALSE;
bFileReaderError := FALSE;

IF nTestStep = 4 THEN
    TEST_FINISHED();
ELSIF tonTimer.Q THEN
    AssertTrue(
        Condition := FALSE,
        Message   := CONCAT(
            CONCAT(
                CONCAT('TestGBSStateMove: timed out at step ', TO_STRING(nTestStep)),
                CONCAT(', eEnumGet=', TO_STRING(TO_UDINT(fbGBS.eEnumGet)))),
            CONCAT(', fActPos=', TO_STRING(fObserved))));
    TEST_FINISHED();
END_IF
END_METHOD

(* In-beam RTD gating test. The two GBS RTDs are vetoed while OUT and active
   in any target state, faulting above the DB reactive temp setpoint (30).
   Rides the state-move test: with temp held high, asserts no fault OUT and a
   fault in a target, then drops the temp and asserts the fault clears. *)
METHOD TestTempFFO
VAR_INST
    tonTimer    : TON;
    nStep       : UINT := 0;
    bOutChecked : BOOL := FALSE;
    bInChecked  : BOOL := FALSE;
END_VAR
VAR CONSTANT
    nLastStep : UINT := 3;
END_VAR
(* Do we fault at the correct times?
   Parasitically depends on the state-move test. *)
TEST('TestGBSTempFFO');

(* Prepare a timeout *)
tonTimer(IN := TRUE, PT := T#10s);

CASE nStep OF
    0:
        (* Set both RTD readings well above the 30 setpoint. *)
        SetGBSTemp(100);
        nStep := nStep + 1;
    1:
        (* Wait to observe both an OUT state (vetoed, no fault) and a
           target state (in beam, fault). *)
        IF fbGBS.eEnumGet = E_GBS_States.OUT THEN
            AssertNeitherTempFault('was in out position');
            bOutChecked := TRUE;
        ELSIF fbGBS.eEnumGet <> E_GBS_States.Unknown THEN
            AssertBothTempFault('was in a target position');
            bInChecked := TRUE;
        END_IF
        IF bOutChecked AND bInChecked THEN
            nStep := nStep + 1;
        END_IF
    2:
        (* Drop both RTD readings below the setpoint again. *)
        SetGBSTemp(0);
        nStep := nStep + 1;
    3:
        AssertNeitherTempFault('has low temp reading');
        nStep := nStep + 1;
END_CASE

IF tonTimer.Q OR nStep > nLastStep THEN
    AssertFalse(tonTimer.Q, 'Timeout in GBS temp FFO test');
    TEST_FINISHED();
END_IF
END_METHOD

END_FUNCTION_BLOCK

// ---- Devices/GBS/FB_GBS.TcPOU
(* Grating Beam Splitter (GBS): thin ND-framework state-mover wrapper.
   Y mover via FB_PositionStatePMPSND (states OUT, TARGET1a/b, TARGET2a/b,
   TARGET3a/b, TARGET4..6), plus a tick site for two in-beam RTDs gated
   on state. Caller-owned deps injected via FB_Init REFERENCE TO and
   forwarded to fbStates; enum bridge and toggles re-forwarded each cycle. *)
{attribute 'call_after_init'}
FUNCTION_BLOCK FB_GBS
VAR_INPUT
    // Set this to a non-unknown value to request a new move.
    {attribute 'pytmc' := '
        pv: MMS:STATE:SET
        io: io
    '}
    eEnumSet : E_GBS_States;
END_VAR
VAR
    {attribute 'pytmc' := 'pv: RTD:01'}
    fbRTD1 : FB_CC_TempSensor;

    {attribute 'pytmc' := 'pv: RTD:02'}
    fbRTD2 : FB_CC_TempSensor;

    (* REFERENCE TO backing fields populated by FB_Init. Same names as
       FB_Init params; THIS^. disambiguates inside FB_Init.
       Live-bound to caller storage for the lifetime of the FB. *)
    {attribute 'no_copy'}
    aiMotionStage         : REFERENCE TO ARRAY[1..MotionConstants.MAX_STATE_MOTORS] OF I_MotionStage;
    {attribute 'no_copy'}
    astPositionState      : REFERENCE TO ARRAY[1..MotionConstants.MAX_STATE_MOTORS]
                                            OF ARRAY[1..GeneralConstants.MAX_STATES] OF ST_PositionState;
    {attribute 'no_copy'}
    fbFFHWO               : REFERENCE TO FB_HardwareFFOutput;
    {attribute 'no_copy'}
    fbArbiter             : REFERENCE TO FB_Arbiter;
    sDeviceName           : STRING;
    sTransitionKey        : STRING;
    bEnableMotion         : BOOL := TRUE;
    bEnableBeamParams     : BOOL;
    bEnablePositionLimits : BOOL;
    bReadDBNow            : BOOL;
    bFileReaderBusy       : REFERENCE TO BOOL;
    bFileReaderError      : REFERENCE TO BOOL;

    (* One configurator per GBS state (OUT + 9 targets). Writes the
       per-state sName and fDelta. Ticked cyclically in the body AFTER
       fbStates so its writes win over the template baseline
       FB_StateSetup applied via FB_CC_StatePMPSConfig. Idempotent once
       stPositionState.bUpdated trips. *)
    afbStateDefaults : ARRAY[1..10] OF FB_CC_InternalStateConfig[
        (stPositionState := astPositionState[1][E_GBS_States.OUT],
         sName           := 'OUT',
         fDelta          := FDELTA_DEFAULT),
        (stPositionState := astPositionState[1][E_GBS_States.TARGET1a],
         sName           := 'TARGET1a',
         fDelta          := FDELTA_DEFAULT),
        (stPositionState := astPositionState[1][E_GBS_States.TARGET1b],
         sName           := 'TARGET1b',
         fDelta          := FDELTA_DEFAULT),
        (stPositionState := astPositionState[1][E_GBS_States.TARGET2a],
         sName           := 'TARGET2a',
         fDelta          := FDELTA_DEFAULT),
        (stPositionState := astPositionState[1][E_GBS_States.TARGET2b],
         sName           := 'TARGET2b',
         fDelta          := FDELTA_DEFAULT),
        (stPositionState := astPositionState[1][E_GBS_States.TARGET3a],
         sName           := 'TARGET3a',
         fDelta          := FDELTA_DEFAULT),
        (stPositionState := astPositionState[1][E_GBS_States.TARGET3b],
         sName           := 'TARGET3b',
         fDelta          := FDELTA_DEFAULT),
        (stPositionState := astPositionState[1][E_GBS_States.TARGET4],
         sName           := 'TARGET4',
         fDelta          := FDELTA_DEFAULT),
        (stPositionState := astPositionState[1][E_GBS_States.TARGET5],
         sName           := 'TARGET5',
         fDelta          := FDELTA_DEFAULT),
        (stPositionState := astPositionState[1][E_GBS_States.TARGET6],
         sName           := 'TARGET6',
         fDelta          := FDELTA_DEFAULT)
    ];

    {attribute 'pytmc' := 'pv: MMS'}
    fbStates : FB_PositionStatePMPSND(
        aiMotionStage         := aiMotionStage,
        astPositionState      := astPositionState,
        nActiveMotorCount     := 1,
        eEnumSet              := eEnumSet,
        eEnumGet              := eEnumGet,
        bEnableMotion         := bEnableMotion,
        eMotionRequestPolicy  := E_MotionRequestPolicy.INTERRUPT,
        bEnableBeamParams     := bEnableBeamParams,
        bEnablePositionLimits := bEnablePositionLimits,
        bReadDBNow            := bReadDBNow,
        bFileReaderBusy       := bFileReaderBusy,
        bFileReaderError      := bFileReaderError,
        fbFFHWO               := fbFFHWO,
        fbArbiter             := fbArbiter,
        sDeviceName           := sDeviceName,
        sTransitionKey        := sTransitionKey
    );
    i : UINT;
END_VAR
VAR_OUTPUT
    // The current position state as an enum.
    {attribute 'pytmc' := '
        pv: MMS:STATE:GET
        io: i
    '}
    eEnumGet: E_GBS_States;
    // The PMPS database lookup associated with the current position state.
    stDbStateParams: ST_DbStateParams;
END_VAR
VAR CONSTANT
    (* GBS-wide default tolerance for state in-position detection,
       applied per-state by afbStateDefaults. *)
    FDELTA_DEFAULT : LREAL := 2;
END_VAR

(* Nil-ref guards: every REFERENCE TO backing field must be bound. *)
IF NOT __ISVALIDREF(aiMotionStage)
   OR NOT __ISVALIDREF(astPositionState)
   OR NOT __ISVALIDREF(fbFFHWO)
   OR NOT __ISVALIDREF(fbArbiter) THEN
    RETURN;
END_IF

(* Device-side per-state defaults (afbStateDefaults) are written
   once in FB_CC_InternalStateConfig.CallAfterInit; no cyclic tick. *)
fbStates(stDbStateParams=> stDbStateParams);

(* In-beam RTDs: only fault when something is actually in the beam
   (i.e. not OUT). Driven by the PMPS DB temp setpoint. *)
fbRTD1(
    fFaultThreshold := fbStates.stDbStateParams.stReactiveParams.nTempSP,
    bVeto           := eEnumGet = E_GBS_States.OUT,
    sDevName        := sDeviceName,
    io_fbFFHWO      := fbFFHWO
);
fbRTD2(
    fFaultThreshold := fbStates.stDbStateParams.stReactiveParams.nTempSP,
    bVeto           := eEnumGet = E_GBS_States.OUT,
    sDevName        := sDeviceName,
    io_fbFFHWO      := fbFFHWO
);

(* Auto-fired after FB_Init. fbStates' inline-init ran first and
   forwarded nil refs, so this re-supplies the now-valid refs via
   fbStates.CallAfterInitStateMover / CallAfterInitPMPS and writes the
   per-state device defaults. *)
{attribute 'call_after_init'}
METHOD CallAfterInit
afbStateDefaults[1].CallAfterInit(stPositionState := THIS^.astPositionState[1][E_GBS_States.OUT]);
afbStateDefaults[2].CallAfterInit(stPositionState := THIS^.astPositionState[1][E_GBS_States.TARGET1a]);
afbStateDefaults[3].CallAfterInit(stPositionState := THIS^.astPositionState[1][E_GBS_States.TARGET1b]);
afbStateDefaults[4].CallAfterInit(stPositionState := THIS^.astPositionState[1][E_GBS_States.TARGET2a]);
afbStateDefaults[5].CallAfterInit(stPositionState := THIS^.astPositionState[1][E_GBS_States.TARGET2b]);
afbStateDefaults[6].CallAfterInit(stPositionState := THIS^.astPositionState[1][E_GBS_States.TARGET3a]);
afbStateDefaults[7].CallAfterInit(stPositionState := THIS^.astPositionState[1][E_GBS_States.TARGET3b]);
afbStateDefaults[8].CallAfterInit(stPositionState := THIS^.astPositionState[1][E_GBS_States.TARGET4]);
afbStateDefaults[9].CallAfterInit(stPositionState := THIS^.astPositionState[1][E_GBS_States.TARGET5]);
afbStateDefaults[10].CallAfterInit(stPositionState := THIS^.astPositionState[1][E_GBS_States.TARGET6]);

THIS^.fbStates.CallAfterInitStateMover(
    aiMotionStage         := aiMotionStage,
    astPositionState      := astPositionState,
    nActiveMotorCount     := 1,
    eEnumSet              := eEnumSet,
    eEnumGet              := eEnumGet,
    bEnableMotion         := bEnableMotion,
    eMotionRequestPolicy  := E_MotionRequestPolicy.INTERRUPT,
);

THIS^.fbStates.CallAfterInitPMPS(
    aiMotionStage         := aiMotionStage,
    astPositionState      := astPositionState,
    bEnableBeamParams     := bEnableBeamParams,
    bEnablePositionLimits := bEnablePositionLimits,
    bReadDBNow            := bReadDBNow,
    bFileReaderBusy       := bFileReaderBusy,
    bFileReaderError      := bFileReaderError,
    fbFFHWO               := fbFFHWO,
    fbArbiter             := fbArbiter,
    sDeviceName           := sDeviceName,
    sTransitionKey        := sTransitionKey
);
END_METHOD

(* Stores FB_Init inputs into instance fields; every non-value input is
   REFERENCE TO, REF= bound for the FB lifetime. fbStates inline-init
   captured these params at construction, so this records the same refs
   on THIS^ for body use and live caller writes. *)
{attribute 'analysis' := '-33'}
METHOD FB_Init : BOOL
VAR_INPUT
    bInitRetains           : BOOL;
    bInCopyCode            : BOOL;
    aiMotionStage          : REFERENCE TO ARRAY[1..MotionConstants.MAX_STATE_MOTORS] OF I_MotionStage;
    astPositionState       : REFERENCE TO ARRAY[1..MotionConstants.MAX_STATE_MOTORS]
                                            OF ARRAY[1..GeneralConstants.MAX_STATES] OF ST_PositionState;
    fbFFHWO                : REFERENCE TO FB_HardwareFFOutput;
    fbArbiter              : REFERENCE TO FB_Arbiter;
    sDeviceName            : STRING;
    sTransitionKey         : STRING;
    bEnableBeamParams      : BOOL;
    bEnablePositionLimits  : BOOL;
    bReadDBNow             : BOOL;
    bFileReaderBusy       : REFERENCE TO BOOL;
    bFileReaderError      : REFERENCE TO BOOL;
END_VAR
THIS^.aiMotionStage    REF= aiMotionStage;
THIS^.astPositionState REF= astPositionState;
THIS^.fbFFHWO          REF= fbFFHWO;
THIS^.fbArbiter        REF= fbArbiter;
THIS^.sDeviceName      := sDeviceName;
THIS^.sTransitionKey   := sTransitionKey;
THIS^.bEnableBeamParams     := bEnableBeamParams;
THIS^.bEnablePositionLimits := bEnablePositionLimits;
THIS^.bReadDBNow            := bReadDBNow;
THIS^.bFileReaderBusy       REF= bFileReaderBusy;
THIS^.bFileReaderError      REF= bFileReaderError;
END_METHOD

END_FUNCTION_BLOCK

// ---- Tests/FB_IPMTest.TcPOU
(* Single integration smoke for FB_IPM. Proves the wrapper wiring (REFERENCE TO
   refs, CallAfterInit chain, fbStates inline-init, per-state defaults, PMPS key
   registration) drives the motor to the configured fPosition for OUT then
   TARGET1, asserting each within fTolerance. State-mover-only device, so no
   temp-FFO test; the motion stack is covered by the motion-abstraction suite. *)
{attribute 'analysis' := '-33'}
FUNCTION_BLOCK FB_IPMTest EXTENDS FB_TestSuite
VAR
    (* Caller-owned axis, persistent storage, and Y motor.
       In a real PRG the AxisRef would come from MAIN.Mxx. *)
    axRef    : ARRAY[1..2] OF AXIS_REF;
    fbPDS    : LCLS_Tc_DevAbs.FB_PersistentDataStorage;

    (* FB_IPM is single-axis (nActiveMotorCount := 1), so only slot 1
       holds a real motor. aiMotionStage is sized to
       MotionConstants.MAX_STATE_MOTORS to match FB_IPM.FB_Init's
       fixed-size signature; slots 2-4 default-init to a nil interface
       and are never touched. *)
    fbMotorX : FB_MotionStageNC(AxisRef := axRef[1], iPersistentDataStorage := fbPDS, sName := 'X');
    fbMotorY : FB_MotionStageNC(AxisRef := axRef[2], iPersistentDataStorage := fbPDS, sName := 'Y');
    aiMotionStage : ARRAY[1..MotionConstants.MAX_STATE_MOTORS] OF I_MotionStage := [fbMotorY];

    {attribute 'pytmc' := '
        pv: MMS
        array: 1..1 | 1..5
    '}
    astPositionState : ARRAY[1..MotionConstants.MAX_STATE_MOTORS]
                         OF ARRAY[1..GeneralConstants.MAX_STATES] OF ST_PositionState;

    fbFFHWO    : FB_HardwareFFOutput;
    fbArbiter  : FB_Arbiter(1);
    fbSubSysIO : FB_DummyArbIO;

    sDeviceName    : STRING := 'TST:IPM';
    sTransitionKey : STRING := 'TST:IPM-TRANSITION';

    (* Caller-owned file-reader status, bound to FB_IPM by REFERENCE
       TO. In a real PRG these point at MOTION_GVL.fbPmpsFileReader;
       here they stay FALSE so the DB read proceeds. *)
    bFileReaderBusy  : BOOL;
    bFileReaderError : BOOL;

    fbIPM : FB_IPM(
        aiMotionStage         := aiMotionStage,
        astPositionState      := astPositionState,
        fbFFHWO               := fbFFHWO,
        fbArbiter             := fbArbiter,
        sDeviceName           := sDeviceName,
        sTransitionKey        := sTransitionKey,
        bEnableBeamParams     := TRUE,
        bEnablePositionLimits := TRUE,
        bReadDBNow            := TRUE,
        bFileReaderBusy       := bFileReaderBusy,
        bFileReaderError      := bFileReaderError
    );

    (* Per-install PMPS-side state config (caller-owned). Mirrors what
       a real PRG_xxL0_IPM would declare. stDefault is the caller-owned
       baseline template that FB_CC_StatePMPSConfig's inner FB_StateSetup
       preloads from; fbIPM subsequently overrides per-state sName and
       fDelta via its own FB_CC_InternalStateConfig array. sPmpsState
       keys match the fake DB seeded by FB_CC_PMPSTestSetup. *)
    stDefault : ST_PositionState := (
        bMoveOk       := TRUE,
        bValid        := TRUE,
        bUseRawCounts := FALSE
    );

    afbStatePMPS : ARRAY[1..5] OF FB_CC_StatePMPSConfig[
        (stPositionState := astPositionState[1][E_IPM_States.OUT],
         stDefault       := stDefault,
         fPosition       := 10,
         sPmpsState      := 'TST:IPM-OUT'),
        (stPositionState := astPositionState[1][E_IPM_States.TARGET1],
         stDefault       := stDefault,
         fPosition       := 20,
         sPmpsState      := 'TST:IPM-TARGET1'),
        (stPositionState := astPositionState[1][E_IPM_States.TARGET2],
         stDefault       := stDefault,
         fPosition       := 30,
         sPmpsState      := 'TST:IPM-TARGET2'),
        (stPositionState := astPositionState[1][E_IPM_States.TARGET3],
         stDefault       := stDefault,
         fPosition       := 40,
         sPmpsState      := 'TST:IPM-TARGET3'),
        (stPositionState := astPositionState[1][E_IPM_States.TARGET4],
         stDefault       := stDefault,
         fPosition       := 50,
         sPmpsState      := 'TST:IPM-TARGET4')
    ];

    bFirstScan : BOOL := TRUE;
    i          : UINT;
END_VAR

TestStateMove();

(* Smoke test for IPM state-move wiring. Walks OUT then TARGET1 and asserts
   each lands within fTolerance of the configured fPosition. Mirrors FB_PPMTest:
   stageReady gate, NOT bMoving + tolerance check per state, 60s watchdog, on
   timeout AssertTrue(FALSE, ...) with the step and observed position. *)
METHOD TestStateMove
VAR_INST
    tonTimer  : TON;
    nTestStep : INT := 0;
    fObserved : LREAL;
END_VAR
VAR CONSTANT
    fTolerance : LREAL := 2.0;
END_VAR
TEST('TestIPMStateMove');

tonTimer(IN := TRUE, PT := T#60s);
fObserved := fbMotorY.stMotionStatus.fActPosition;

CASE nTestStep OF
    0:
        IF bFirstScan THEN
            fbMotorY.SetModeEnableLimits(
                LimBackward    := TRUE,
                LimForward     := TRUE,
                HomeEnable     := FALSE,
                BrakeMode      := E_StageBrakeMode.IF_ENABLED,
                EnableMode     := E_StageEnableMode.DURING_MOTION,
                HomeMode       := E_EpicsHomeCmd.LOW_LIMIT,
                UserEnable     := TRUE,
                HardwareEnable := TRUE
            );
            fbMotorX.SetModeEnableLimits(
                LimBackward    := TRUE,
                LimForward     := TRUE,
                HomeEnable     := FALSE,
                BrakeMode      := E_StageBrakeMode.IF_ENABLED,
                EnableMode     := E_StageEnableMode.DURING_MOTION,
                HomeMode       := E_EpicsHomeCmd.LOW_LIMIT,
                UserEnable     := TRUE,
                HardwareEnable := TRUE
            );
            fbMotorX.SetVelocity(Velocity := 15.5);
            fbMotorX.RestoreMotionParams      := FALSE;
            fbMotorX.DoNotRestoreNcParameters := TRUE;
            fbMotorY.SetVelocity(Velocity := 15.5);
            fbMotorY.RestoreMotionParams      := FALSE;
            fbMotorY.DoNotRestoreNcParameters := TRUE;
            bFileReaderBusy  := TRUE;
            bFileReaderError := FALSE;
            bFirstScan := FALSE;
        END_IF
        nTestStep      := 1;
    1:
        IF fbMotorY.stMotionStatus.bStageReady
           AND NOT fbMotorY.stMotionStatus.bError THEN
            fbIPM.eEnumSet := E_IPM_States.OUT;
            nTestStep      := 2;
        END_IF
    2:
        (* OUT is configured at fPosition := 10 in afbStatePMPS[1]. *)
        IF fbIPM.eEnumGet = E_IPM_States.OUT
           AND NOT fbMotorY.stMotionStatus.bMoving
           AND ABS(fObserved - 10.0) <= fTolerance THEN
            fbIPM.eEnumSet := E_IPM_States.TARGET1;
            nTestStep      := 3;
        END_IF
    3:
        (* TARGET1 is configured at fPosition := 20 in afbStatePMPS[2]. *)
        IF fbIPM.eEnumGet = E_IPM_States.TARGET1
           AND NOT fbMotorY.stMotionStatus.bMoving
           AND ABS(fObserved - 20.0) <= fTolerance THEN
            AssertTrue(
                Condition := TRUE,
                Message   := 'TestIPMStateMove: OUT then TARGET1 reached within tolerance');
            nTestStep := 4;
        END_IF
END_CASE

(* Fake PMPS handling. *)
fbSubSysIO(
    LA  := fbArbiter,
    FFO := fbFFHWO
);

fbPDS();
fbMotorY();
fbIPM();

bFileReaderBusy  := FALSE;
bFileReaderError := FALSE;

IF nTestStep = 4 THEN
    TEST_FINISHED();
ELSIF tonTimer.Q THEN
    AssertTrue(
        Condition := FALSE,
        Message   := CONCAT(
            CONCAT(
                CONCAT('TestIPMStateMove: timed out at step ', TO_STRING(nTestStep)),
                CONCAT(', eEnumGet=', TO_STRING(TO_UDINT(fbIPM.eEnumGet)))),
            CONCAT(', fActPos=', TO_STRING(fObserved))));
    TEST_FINISHED();
END_IF
END_METHOD

END_FUNCTION_BLOCK

// ---- Devices/IPM/FB_IPM.TcPOU
(* Intensity Profile Monitor (IPM): thin ND-framework state-mover wrapper.
   Y mover via FB_PositionStatePMPSND (states OUT, TARGET1..TARGET4).
   Caller-owned motors, stage/state arrays, fast-fault and arbiter are
   injected via FB_Init REFERENCE TO and forwarded to fbStates; enum
   bridge and toggles re-forwarded each cycle. *)
{attribute 'call_after_init'}
FUNCTION_BLOCK FB_IPM
VAR_INPUT
    // Set this to a non-unknown value to request a new move.
    {attribute 'pytmc' := '
        pv: MMS:STATE:SET
        io: io
    '}
    eEnumSet : E_IPM_States;
END_VAR
VAR
    (* REFERENCE TO backing fields populated by FB_Init. Same names as
       FB_Init params; THIS^. disambiguates inside FB_Init.
       Live-bound to caller storage for the lifetime of the FB. *)
    {attribute 'no_copy'}
    aiMotionStage         : REFERENCE TO ARRAY[1..MotionConstants.MAX_STATE_MOTORS] OF I_MotionStage;
    {attribute 'no_copy'}
    astPositionState      : REFERENCE TO ARRAY[1..MotionConstants.MAX_STATE_MOTORS]
                                            OF ARRAY[1..GeneralConstants.MAX_STATES] OF ST_PositionState;
    {attribute 'no_copy'}
    fbFFHWO               : REFERENCE TO FB_HardwareFFOutput;
    {attribute 'no_copy'}
    fbArbiter             : REFERENCE TO FB_Arbiter;
    sDeviceName           : STRING;
    sTransitionKey        : STRING;
    bEnableMotion         : BOOL := TRUE;
    bEnableBeamParams     : BOOL;
    bEnablePositionLimits : BOOL;
    bReadDBNow            : BOOL;

    bFileReaderBusy       : REFERENCE TO BOOL;
    bFileReaderError      : REFERENCE TO BOOL;

